fbFilterWeight2(
				rIn:=				DINT_TO_REAL(InWeight2Value), 
				tTimeConstant:= 	T#25MS, //bylo 25
				rOut=>				rFilteredWeight2Value);
				
fbFilterWeight3(
				rIn:=				DINT_TO_REAL(InWeight3Value), 
				tTimeConstant:= 	T#52MS, //bylo 25
				rOut=>				rFilteredWeight3Value);
				
fbFilterWeight4(
				rIn:=				DINT_TO_REAL(InWeight4Value), 
				tTimeConstant:= 	T#25MS, //bylo 25
				rOut=>				rFilteredWeight4Value);
///////////////////////////////////////////////////////////////////////////////				
fbFilterWeight5(
				rIn:=				DINT_TO_REAL(InWeight5Value), 
				tTimeConstant:= 	T#25MS, //bylo 25
				rOut=>				rFilteredWeight5Value);
								
fbFilterWeight6(
				rIn:=				DINT_TO_REAL(InWeight6Value), 
				tTimeConstant:= 	T#25MS, //bylo 25
				rOut=>				rFilteredWeight6Value);														
/////////////////////////////////////////////////////////////////////////////

tonIbWeight1FormSensor			(IN:=IbWeight1FormSensor ,		PT:=T#120MS); //160
tonIbWeight2FormSensor			(IN:=IbWeight2FormSensor ,		PT:=T#120MS); //160
tonIbWeight3FormSensor			(IN:=IbWeight3FormSensor ,		PT:=T#120MS); //160
tonIbWeight4FormSensor			(IN:=IbWeight4FormSensor ,		PT:=T#120MS); //160
tonIbWeight5FormSensor			(IN:=IbWeight5FormSensor ,		PT:=T#120MS); //60
tonIbWeight6FormSensor			(IN:=IbWeight6FormSensor ,		PT:=T#120MS); //60

IF VIS.nFormTransportersScrewerVelocitySVShow < 500 THEN
	fbIbWeight1FormBeforeSensor	(bIN:=IbWeight1ActuatorSensorUp,	tFilterTimeOn:=T#70MS,	tFilterTimeOff:=T#150MS);
	fbIbWeight2FormBeforeSensor	(bIN:=IbWeight2ActuatorSensorUp,	tFilterTimeOn:=T#70MS,	tFilterTimeOff:=T#150MS);
	fbIbWeight3FormBeforeSensor	(bIN:=IbWeight3ActuatorSensorUp,	tFilterTimeOn:=T#70MS,	tFilterTimeOff:=T#150MS);
	fbIbWeight4FormBeforeSensor	(bIN:=IbWeight4ActuatorSensorUp,	tFilterTimeOn:=T#70MS,	tFilterTimeOff:=T#150MS);
ELSE
	fbIbWeight1FormBeforeSensor	(bIN:=IbWeight1ActuatorSensorUp,	tFilterTimeOn:=T#10MS,	tFilterTimeOff:=T#10MS);//bylo 40 i 20
	fbIbWeight2FormBeforeSensor	(bIN:=IbWeight2ActuatorSensorUp,	tFilterTimeOn:=T#10MS,	tFilterTimeOff:=T#10MS);//bylo 40 i 20
	fbIbWeight3FormBeforeSensor	(bIN:=IbWeight3ActuatorSensorUp,	tFilterTimeOn:=T#10MS,	tFilterTimeOff:=T#10MS);//bylo 40 i 20
	fbIbWeight4FormBeforeSensor	(bIN:=IbWeight4ActuatorSensorUp,	tFilterTimeOn:=T#10MS,	tFilterTimeOff:=T#10MS);//bylo 40 i 20	
END_IF

IF VIS.nFormTransportersDispencerVelocitySVShow < 500 THEN
	fbIbWeight5FormBeforeSensor	(bIN:=IbWeight5FormSensor,			tFilterTimeOn:=T#70MS,	tFilterTimeOff:=T#150MS);
	fbIbWeight6FormBeforeSensor	(bIN:=IbWeight6FormSensor,			tFilterTimeOn:=T#70MS,	tFilterTimeOff:=T#150MS);
ELSE
	fbIbWeight5FormBeforeSensor	(bIN:=IbWeight5FormSensor,			tFilterTimeOn:=T#70MS,	tFilterTimeOff:=T#150MS);
	fbIbWeight6FormBeforeSensor	(bIN:=IbWeight6FormSensor,			tFilterTimeOn:=T#70MS,	tFilterTimeOff:=T#150MS);
END_IF
END_ACTION

ACTION aWeight1:
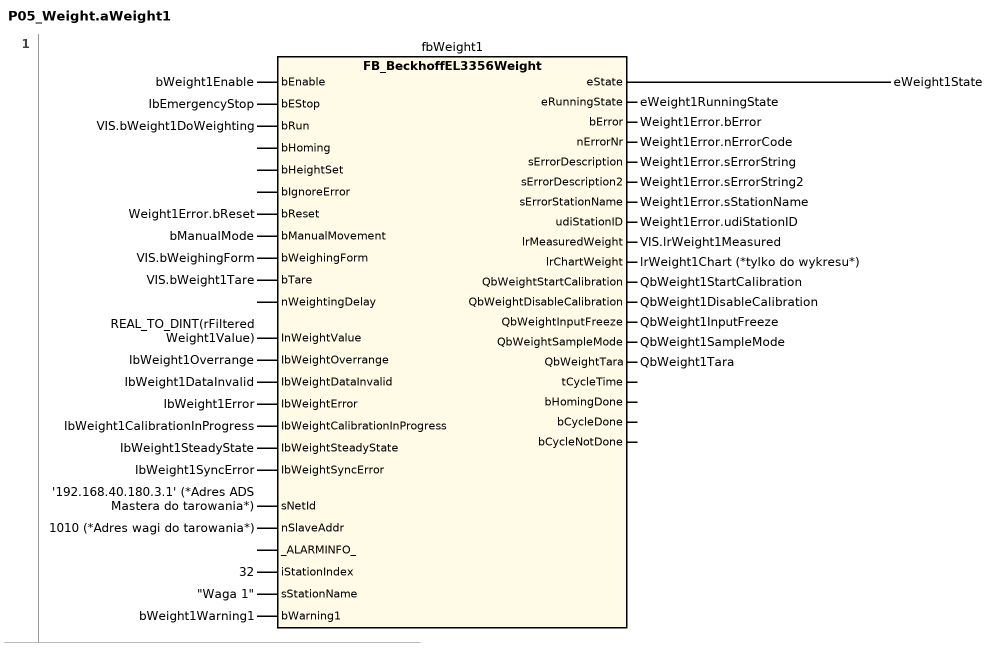
// NETWORK 1
fbWeight1(
    bEnable := bWeight1Enable,
    bEStop := IbEmergencyStop,
    bRun := VIS.bWeight1DoWeighting,
    bReset := Weight1Error.bReset,
    bManualMovement := bManualMode,
    bWeighingForm := VIS.bWeighingForm,
    bTare := VIS.bWeight1Tare,
    InWeightValue := REAL_TO_DINT(rFilteredWeight1Value),
    IbWeightOverrange := IbWeight1Overrange,
    IbWeightDataInvalid := IbWeight1DataInvalid,
    IbWeightError := IbWeight1Error,
    IbWeightCalibrationInProgress := IbWeight1CalibrationInProgress,
    IbWeightSteadyState := IbWeight1SteadyState,
    IbWeightSyncError := IbWeight1SyncError,
    sNetId := '192.168.40.180.3.1' (*Adres ADS Mastera do tarowania*),
    nSlaveAddr := 1010 (*Adres wagi do tarowania*),
    iStationIndex := 32,
    sStationName := "Waga 1",
    bWarning1 := bWeight1Warning1,
    eRunningState => eWeight1RunningState,
    bError => Weight1Error.bError,
    nErrorNr => Weight1Error.nErrorCode,
    sErrorDescription => Weight1Error.sErrorString,
    sErrorDescription2 => Weight1Error.sErrorString2,
    sErrorStationName => Weight1Error.sStationName,
    udiStationID => Weight1Error.udiStationID,
    lrMeasuredWeight => VIS.lrWeight1Measured,
    lrChartWeight => lrWeight1Chart (*tylko do wykresu*),
    QbWeightStartCalibration => QbWeight1StartCalibration,
    QbWeightDisableCalibration => QbWeight1DisableCalibration,
    QbWeightInputFreeze => QbWeight1InputFreeze,
    QbWeightSampleMode => QbWeight1SampleMode,
    QbWeightTara => QbWeight1Tara); // FB_BeckhoffEL3356Weight
eWeight1State := fbWeight1.eState;
END_ACTION

ACTION aWeight2:
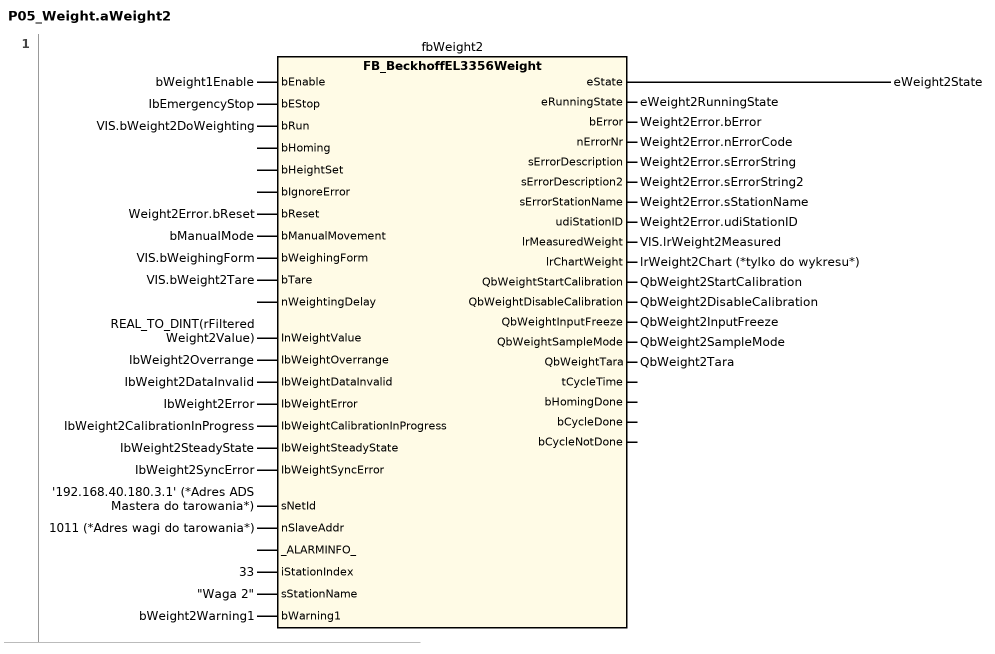
// NETWORK 1
fbWeight2(
    bEnable := bWeight1Enable,
    bEStop := IbEmergencyStop,
    bRun := VIS.bWeight2DoWeighting,
    bReset := Weight2Error.bReset,
    bManualMovement := bManualMode,
    bWeighingForm := VIS.bWeighingForm,
    bTare := VIS.bWeight2Tare,
    InWeightValue := REAL_TO_DINT(rFilteredWeight2Value),
    IbWeightOverrange := IbWeight2Overrange,
    IbWeightDataInvalid := IbWeight2DataInvalid,
    IbWeightError := IbWeight2Error,
    IbWeightCalibrationInProgress := IbWeight2CalibrationInProgress,
    IbWeightSteadyState := IbWeight2SteadyState,
    IbWeightSyncError := IbWeight2SyncError,
    sNetId := '192.168.40.180.3.1' (*Adres ADS Mastera do tarowania*),
    nSlaveAddr := 1011 (*Adres wagi do tarowania*),
    iStationIndex := 33,
    sStationName := "Waga 2",
    bWarning1 := bWeight2Warning1,
    eRunningState => eWeight2RunningState,
    bError => Weight2Error.bError,
    nErrorNr => Weight2Error.nErrorCode,
    sErrorDescription => Weight2Error.sErrorString,
    sErrorDescription2 => Weight2Error.sErrorString2,
    sErrorStationName => Weight2Error.sStationName,
    udiStationID => Weight2Error.udiStationID,
    lrMeasuredWeight => VIS.lrWeight2Measured,
    lrChartWeight => lrWeight2Chart (*tylko do wykresu*),
    QbWeightStartCalibration => QbWeight2StartCalibration,
    QbWeightDisableCalibration => QbWeight2DisableCalibration,
    QbWeightInputFreeze => QbWeight2InputFreeze,
    QbWeightSampleMode => QbWeight2SampleMode,
    QbWeightTara => QbWeight2Tara); // FB_BeckhoffEL3356Weight
eWeight2State := fbWeight2.eState;
END_ACTION

ACTION aWeight3:
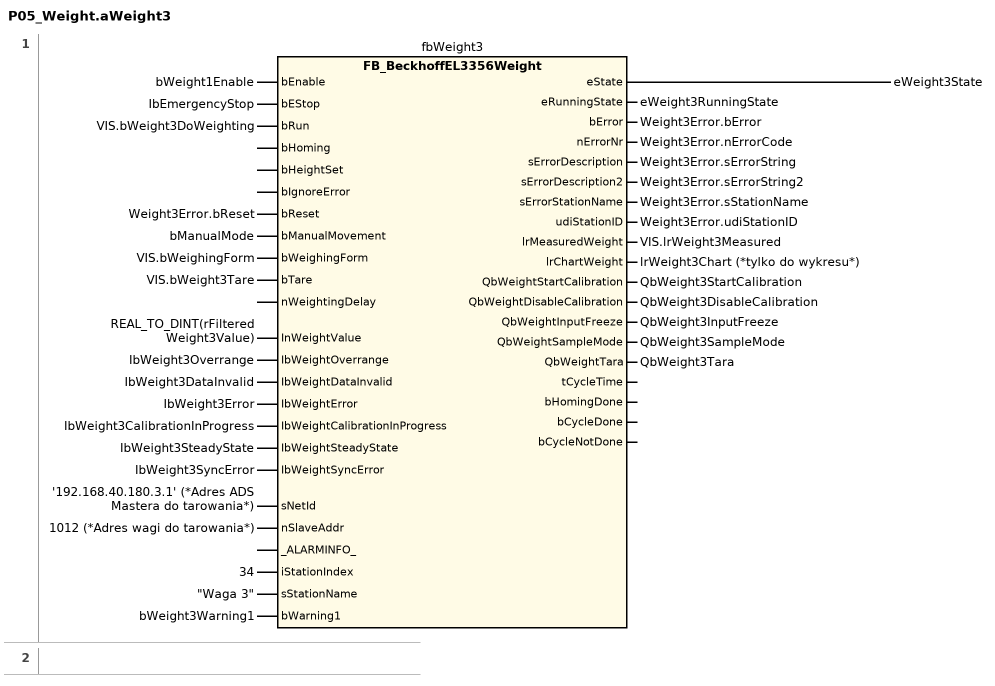
// NETWORK 1
fbWeight3(
    bEnable := bWeight1Enable,
    bEStop := IbEmergencyStop,
    bRun := VIS.bWeight3DoWeighting,
    bReset := Weight3Error.bReset,
    bManualMovement := bManualMode,
    bWeighingForm := VIS.bWeighingForm,
    bTare := VIS.bWeight3Tare,
    InWeightValue := REAL_TO_DINT(rFilteredWeight3Value),
    IbWeightOverrange := IbWeight3Overrange,
    IbWeightDataInvalid := IbWeight3DataInvalid,
    IbWeightError := IbWeight3Error,
    IbWeightCalibrationInProgress := IbWeight3CalibrationInProgress,
    IbWeightSteadyState := IbWeight3SteadyState,
    IbWeightSyncError := IbWeight3SyncError,
    sNetId := '192.168.40.180.3.1' (*Adres ADS Mastera do tarowania*),
    nSlaveAddr := 1012 (*Adres wagi do tarowania*),
    iStationIndex := 34,
    sStationName := "Waga 3",
    bWarning1 := bWeight3Warning1,
    eRunningState => eWeight3RunningState,
    bError => Weight3Error.bError,
    nErrorNr => Weight3Error.nErrorCode,
    sErrorDescription => Weight3Error.sErrorString,
    sErrorDescription2 => Weight3Error.sErrorString2,
    sErrorStationName => Weight3Error.sStationName,
    udiStationID => Weight3Error.udiStationID,
    lrMeasuredWeight => VIS.lrWeight3Measured,
    lrChartWeight => lrWeight3Chart (*tylko do wykresu*),
    QbWeightStartCalibration => QbWeight3StartCalibration,
    QbWeightDisableCalibration => QbWeight3DisableCalibration,
    QbWeightInputFreeze => QbWeight3InputFreeze,
    QbWeightSampleMode => QbWeight3SampleMode,
    QbWeightTara => QbWeight3Tara); // FB_BeckhoffEL3356Weight
eWeight3State := fbWeight3.eState;

// NETWORK 2
END_ACTION

ACTION aWeight4:
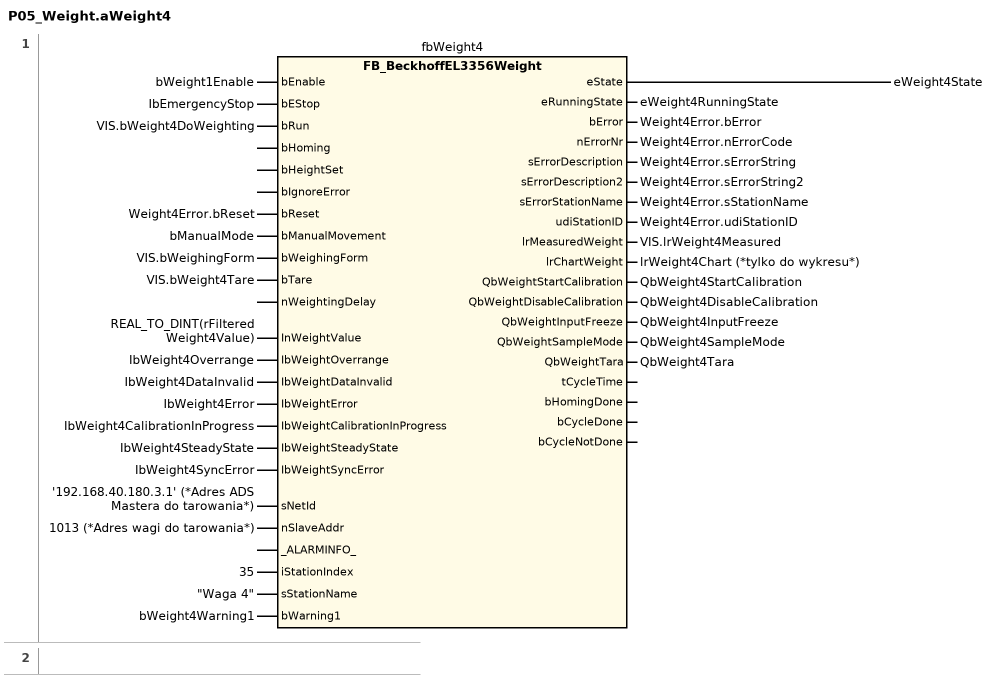
// NETWORK 1
fbWeight4(
    bEnable := bWeight1Enable,
    bEStop := IbEmergencyStop,
    bRun := VIS.bWeight4DoWeighting,
    bReset := Weight4Error.bReset,
    bManualMovement := bManualMode,
    bWeighingForm := VIS.bWeighingForm,
    bTare := VIS.bWeight4Tare,
    InWeightValue := REAL_TO_DINT(rFilteredWeight4Value),
    IbWeightOverrange := IbWeight4Overrange,
    IbWeightDataInvalid := IbWeight4DataInvalid,
    IbWeightError := IbWeight4Error,
    IbWeightCalibrationInProgress := IbWeight4CalibrationInProgress,
    IbWeightSteadyState := IbWeight4SteadyState,
    IbWeightSyncError := IbWeight4SyncError,
    sNetId := '192.168.40.180.3.1' (*Adres ADS Mastera do tarowania*),
    nSlaveAddr := 1013 (*Adres wagi do tarowania*),
    iStationIndex := 35,
    sStationName := "Waga 4",
    bWarning1 := bWeight4Warning1,
    eRunningState => eWeight4RunningState,
    bError => Weight4Error.bError,
    nErrorNr => Weight4Error.nErrorCode,
    sErrorDescription => Weight4Error.sErrorString,
    sErrorDescription2 => Weight4Error.sErrorString2,
    sErrorStationName => Weight4Error.sStationName,
    udiStationID => Weight4Error.udiStationID,
    lrMeasuredWeight => VIS.lrWeight4Measured,
    lrChartWeight => lrWeight4Chart (*tylko do wykresu*),
    QbWeightStartCalibration => QbWeight4StartCalibration,
    QbWeightDisableCalibration => QbWeight4DisableCalibration,
    QbWeightInputFreeze => QbWeight4InputFreeze,
    QbWeightSampleMode => QbWeight4SampleMode,
    QbWeightTara => QbWeight4Tara); // FB_BeckhoffEL3356Weight
eWeight4State := fbWeight4.eState;

// NETWORK 2
END_ACTION

ACTION aWeight5:
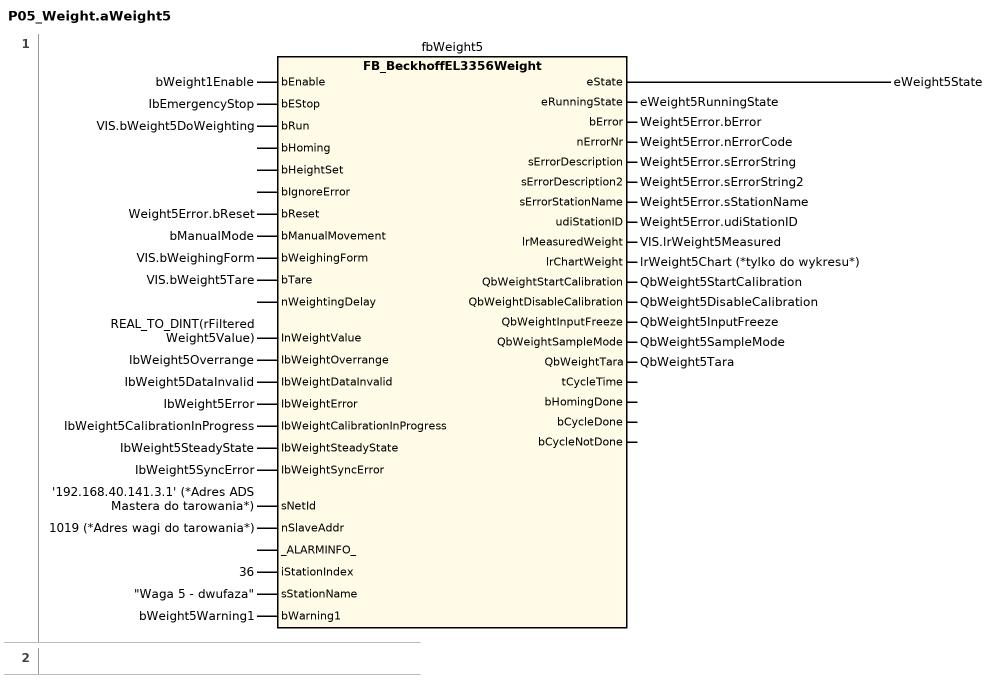
// NETWORK 1
fbWeight5(
    bEnable := bWeight1Enable,
    bEStop := IbEmergencyStop,
    bRun := VIS.bWeight5DoWeighting,
    bReset := Weight5Error.bReset,
    bManualMovement := bManualMode,
    bWeighingForm := VIS.bWeighingForm,
    bTare := VIS.bWeight5Tare,
    InWeightValue := REAL_TO_DINT(rFilteredWeight5Value),
    IbWeightOverrange := IbWeight5Overrange,
    IbWeightDataInvalid := IbWeight5DataInvalid,
    IbWeightError := IbWeight5Error,
    IbWeightCalibrationInProgress := IbWeight5CalibrationInProgress,
    IbWeightSteadyState := IbWeight5SteadyState,
    IbWeightSyncError := IbWeight5SyncError,
    sNetId := '192.168.40.141.3.1' (*Adres ADS Mastera do tarowania*),
    nSlaveAddr := 1019 (*Adres wagi do tarowania*),
    iStationIndex := 36,
    sStationName := "Waga 5 - dwufaza",
    bWarning1 := bWeight5Warning1,
    eRunningState => eWeight5RunningState,
    bError => Weight5Error.bError,
    nErrorNr => Weight5Error.nErrorCode,
    sErrorDescription => Weight5Error.sErrorString,
    sErrorDescription2 => Weight5Error.sErrorString2,
    sErrorStationName => Weight5Error.sStationName,
    udiStationID => Weight5Error.udiStationID,
    lrMeasuredWeight => VIS.lrWeight5Measured,
    lrChartWeight => lrWeight5Chart (*tylko do wykresu*),
    QbWeightStartCalibration => QbWeight5StartCalibration,
    QbWeightDisableCalibration => QbWeight5DisableCalibration,
    QbWeightInputFreeze => QbWeight5InputFreeze,
    QbWeightSampleMode => QbWeight5SampleMode,
    QbWeightTara => QbWeight5Tara); // FB_BeckhoffEL3356Weight
eWeight5State := fbWeight5.eState;

// NETWORK 2
END_ACTION

ACTION aWeight6:
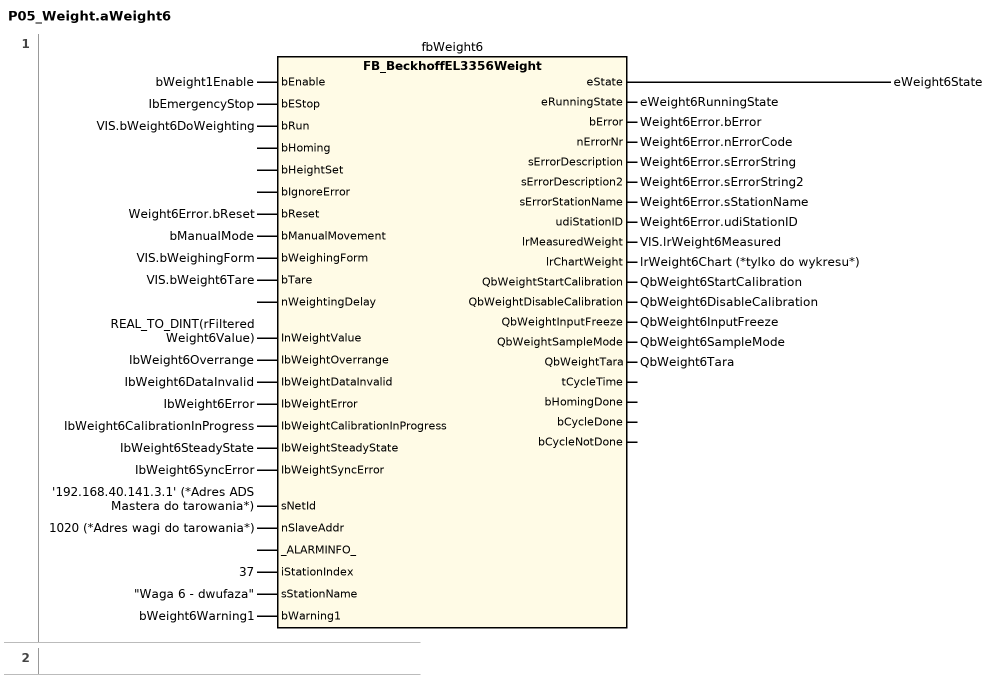
// NETWORK 1
fbWeight6(
    bEnable := bWeight1Enable,
    bEStop := IbEmergencyStop,
    bRun := VIS.bWeight6DoWeighting,
    bReset := Weight6Error.bReset,
    bManualMovement := bManualMode,
    bWeighingForm := VIS.bWeighingForm,
    bTare := VIS.bWeight6Tare,
    InWeightValue := REAL_TO_DINT(rFilteredWeight6Value),
    IbWeightOverrange := IbWeight6Overrange,
    IbWeightDataInvalid := IbWeight6DataInvalid,
    IbWeightError := IbWeight6Error,
    IbWeightCalibrationInProgress := IbWeight6CalibrationInProgress,
    IbWeightSteadyState := IbWeight6SteadyState,
    IbWeightSyncError := IbWeight6SyncError,
    sNetId := '192.168.40.141.3.1' (*Adres ADS Mastera do tarowania*),
    nSlaveAddr := 1020 (*Adres wagi do tarowania*),
    iStationIndex := 37,
    sStationName := "Waga 6 - dwufaza",
    bWarning1 := bWeight6Warning1,
    eRunningState => eWeight6RunningState,
    bError => Weight6Error.bError,
    nErrorNr => Weight6Error.nErrorCode,
    sErrorDescription => Weight6Error.sErrorString,
    sErrorDescription2 => Weight6Error.sErrorString2,
    sErrorStationName => Weight6Error.sStationName,
    udiStationID => Weight6Error.udiStationID,
    lrMeasuredWeight => VIS.lrWeight6Measured,
    lrChartWeight => lrWeight6Chart (*tylko do wykresu*),
    QbWeightStartCalibration => QbWeight6StartCalibration,
    QbWeightDisableCalibration => QbWeight6DisableCalibration,
    QbWeightInputFreeze => QbWeight6InputFreeze,
    QbWeightSampleMode => QbWeight6SampleMode,
    QbWeightTara => QbWeight6Tara); // FB_BeckhoffEL3356Weight
eWeight6State := fbWeight6.eState;

// NETWORK 2
END_ACTION

END_PROGRAM

// ---- POUs/FB/FB_BeckhoffEL3356Weight.TcPOU
(*
Nazwa:			FB_BeckhoffEL3356Weight
Opis:			Obsługa wagi
Wersja:			v0.1
Data:			2019-10-09
Autor:			DP
Urzadzenia:		waga Beckhoff
Konfiguracja:	
Info: 
- podlaczenie po module EL3356-0010
Nastawy modułu "Settings" 
Mode of operation: Standard (INT32)
RMB DATA 
Zaznaczone tylko 
	-Mode0 Filter enable: Dynamic IIR z wartością 0.2
	-Symetric reference potential active
Kalibracja zrobionia z jakaś wagą np 1kg, to wpisane 10000
Gain:1,Rated Output 0.062372, ZeroBalance 0.0209,
ScaleFactor:1, SteadyStateWindow:100ms, CalibrationInterwal:180s
SteadyStateTolerance:10,TestInteval:10,

*)


FUNCTION_BLOCK FB_BeckhoffEL3356Weight
VAR_INPUT
	bEnable: BOOL;						//Zezwolenie na pracę
	bEStop:BOOL;						//Stop Awaryjny włączony
	bRun:BOOL;							//Rozkaz łapania 
	bHoming:BOOL;						//Zezwolenie na wykonanie bazowania i pozycjonowania podajnika
	bHeightSet:BOOL;					//Ustaw wysokość
	bIgnoreError:BOOL;					//Ignorowania błędów cyklu pracy
	bReset:BOOL;						//Reset błędu, jeśli w stanie "eError"
	bManualMovement:BOOL;				//Zezwolenie na ruchy ręcznę
	bWeighingForm: BOOL;				//Wlaczone przewazanie, dluzsze czasy		
	bTare:BOOL;							//Tarowanie Wagi
	nWeightingDelay:UINT;				//Opoźnienie ważenia
	InWeightValue: DINT;				// Wartość wagi
	IbWeightOverrange: BOOL;						
	IbWeightDataInvalid: BOOL;		
	IbWeightError: BOOL;	
	IbWeightCalibrationInProgress: BOOL;
	IbWeightSteadyState: BOOL;
	IbWeightSyncError: BOOL;	
	sNetId:STRING;
	nSlaveAddr:UINT;
	
	_ALARMINFO_ :BOOL;
	iStationIndex:UDINT;					//Numer stacji 
	sStationName:WSTRING;					//Nazwa stacji	

END_VAR
VAR_OUTPUT
	eState: E_Station;						//Stan ogólny bloku
	eRunningState: E_WeightState;			//Stan wewnętrzny
	bError: BOOL;							//Błąd stacji
	nErrorNr: UDINT;						//Nr błędu podajnika platynek
	sErrorDescription:STRING;				//Opis błędu
	sErrorDescription2: STRING;				//Opis błędu 2
	sErrorStationName:STRING;				//Nazwa stacji
	udiStationID:UDINT;						// Nr stacji

	lrMeasuredWeight: LREAL; 				//Zmierzona waga 
	lrChartWeight: LREAL; 					//Zmierzona waga do wykresu
	QbWeightStartCalibration: BOOL;
	QbWeightDisableCalibration: BOOL;
	QbWeightInputFreeze: BOOL;
	QbWeightSampleMode: BOOL;
	QbWeightTara: BOOL;
	tCycleTime:TIME;
	bHomingDone:BOOL;						//Wymagane ponowne bazowanie (blad podczas bazowania lub stop awaryjny)
	bCycleDone:BOOL;
	bCycleNotDone:BOOL;
END_VAR
VAR
	(*Opóźnianie ważenia*)
	tonWeightingDelay: TON;
	
	(*Tarowanie*)
	rtrigTare: R_TRIG;
	
	(*Statystyki*)
	rtrigCycleTimerRead: R_TRIG;
	tonCycleTimer: TON;
	
	(*Próbkowanie wagi*)
	lrMeasuredWeightSampling: LREAL;
	lrWeightSampling: LREAL;
	tonWeightingDoneIfNotSteadyState: TON;
	nWeightingDoneIfNotSteadyState: INT; //Licznik ilości prawdopodobnie błędnych pomiarów
	tonWeightingDoneIfNotSteadyStateReset: TON; // Do resetowania błędu ilości błędnych pomiarów
	//
	tonOverrange	:TON;
	tonError		:TON;	
	
	(*TAROWANIE EEPROM*)
	fbCoE:FB_EcCoESdoWrite;
	wCoeData:WORD;

	nWarCheck1: INT;
	nWarCheck2: INT;
	bMinMaxAvg: BOOL;
	lrMeasuredWeightMax: LREAL;
	lrMeasuredWeightMin: LREAL;

	eLastState: E_Station;							//Stan ogólny bloku
	eLastRunningState: E_WeightState;			//Stan podbloku
	eLastStateTemp: E_Station;						//Stan ogólny bloku
	eLastRunningStateTemp: E_WeightState;		//Stan podbloku
	bStateError: BOOL;
	
	fbCalibrationDisableOff	: FB_InputFilter;

	tWeightingTime: TIME;
	
	//Zmienne od EVENTLOGGER
	bAlarmInit 						: BOOL := TRUE; 
	nAlarmNumerator					: INT;
	arfbAlarm						: ARRAY[0..19] OF  FB_TcAlarm;		//Tablica bloczków błędów
	fbSourceInfo 					: FB_TcSourceInfo;
	iSourceInfo						: I_TcSourceInfo;
	sAlarmTest						: STRING;
	tonEventLogger					: TON;
	//Koniec zmiennych od EVENTLOGGER
END_VAR

VAR_IN_OUT
	bWarning1: BOOL;		//Ostrzezenie przed brakiem stabilizacji wagi
END_VAR

aWeighingForm();
ErrorHandling();
Control();
Statistics();
aStationID();

(*Zapisywanie ostatniego stanu*)
IF eLastStateTemp<>eState THEN
	eLastState := eLastStateTemp;
END_IF
eLastStateTemp := eState;
IF eLastRunningStateTemp<>eRunningState THEN
	eLastRunningState := eLastRunningStateTemp;
END_IF
eLastRunningStateTemp := eRunningState;
(*Koniec Zapisywanie ostatniego stanu*)

//do testów, bo co 180s robi samokalibracje!
fbCalibrationDisableOff(bIN:=bRun, tFilterTimeOn:=T#10MS, tFilterTimeOff:=T#2S);
IF fbCalibrationDisableOff.bOUT THEN
	QbWeightDisableCalibration:=TRUE;
ELSE 
	QbWeightDisableCalibration:=FALSE;
	
END_IF
//QbWeightTara:=bTare;

ACTION aStationID:
udiStationID	:=	iStationIndex;
END_ACTION

ACTION aWeighingForm:
(*
IF bWeighingForm THEN //Wlaczone przewazanie formatek
	nWeightingDelay := 2000; //Opoznienie przed wazeniem
	tWeightingTime	:= T#800MS; //Czas ważenia
ELSE				// Wylaczone przewazanie
	tWeightingTime := T#500MS; //Czas ważenia
END_IF
*)





IF bWeighingForm THEN //Wlaczone przewazanie formatek
	nWeightingDelay := 685;//685 //Opoznienie przed wazeniem
	tWeightingTime	:= T#300MS;//T#150MS; //Czas ważenia
ELSE				// Wylaczone przewazanie
	tWeightingTime := T#150MS;//T#150MS; //Czas ważenia
	//tWeightingTime := T#100MS;//T#490MS;//T#500MS; //Czas ważenia	
END_IF
END_ACTION

ACTION Control:

	(** TIMERY**)
	//Opóźnienie ważenia, trzeba tutaj uwzględnić jeszcze czas ustawiania bitu SteadyState
	tonWeightingDelay(IN:=(eRunningState=E_WeightState.eWeighting), PT:=UINT_TO_TIME(nWeightingDelay));
	//Jeżeli nie ma stabilizacji wagi to po tym czasie podaj pomiar z próbkowania
	tonWeightingDoneIfNotSteadyState(IN:=eRunningState=E_WeightState.eWeighting AND tonWeightingDelay.Q, PT:=tWeightingTime); //bylo 550

	(*****Wyłączenie enable*****)
	IF NOT bEnable THEN
		IF eState <> E_Station.eDisabled AND eState <> E_Station.ePreparingToDisable THEN
				eState 				:= E_Station.ePreparingToDisable; 
		END_IF	
	END_IF

	(*****Estop*****)
	IF NOT bEstop  THEN	
		IF eState <> E_Station.eAborted AND eState <> E_Station.eAborting AND eState <> E_Station.eDisabled THEN
				eState 				:= E_Station.eAborting; 
		END_IF
	END_IF

	CASE eState OF
	/////////////////////////////	
		E_Station.eDisabled: 					// Stan nieaktywnosci (Stacja wyłączona) 

			IF bEnable THEN
				eState 				:= E_Station.ePreparingToReady; 
			END_IF 
			
    /////////////////////////////	    
		E_Station.eAborted: 					// Stan bezpiecznego zatrzymania (po Abortingu) 

			IF bEStop THEN
				eState 				:= E_Station.ePreparingToReady;
			END_IF
			
	/////////////////////////////	
		E_Station.eAborting:                 	// Stan bezpiecznego zatrzymywania (po EStopie)

		
			eState := E_Station.eAborted;  
			eRunningState:=E_WeightState.eDisabled;
			
	/////////////////////////////			
		E_Station.eError:                 	 	// Stan błędu 	

			IF bReset THEN
				eState 				:= E_Station.eResetting;
				
			END_IF
						
	/////////////////////////////
		E_Station.eResetting:					// Stan resetowania bledu (po Errorze)
	
			bError := FALSE;

			IF NOT bError THEN
				nErrorNr 			:=	0;
   				sErrorDescription 	:=	'';
				eState 				:=	E_Station.ePreparingToReady;
			ELSE
				eState 				:=	E_Station.eError;
			END_IF
        
	/////////////////////////////
		E_Station.eManualMovement:     			// Stan ruchów manualnych  

			ManualMovements();
			//Wyjście z trybu serwisowego
			IF NOT bManualMovement THEN
				eState:=E_Station.eReady;
			END_IF

	/////////////////////////////
		E_Station.eHoming:						// Stan bazowania 

			Homing();
			IF NOT bHoming AND NOT bHeightSet THEN
			   eState:=E_Station.ePreparingToReady;
			END_IF		
			
	/////////////////////////////
		E_Station.eHomingDone:                  // Stan wykonania bazowania 
	
			bHomingDone							:=	TRUE;
			IF NOT bHoming AND NOT bHeightSet THEN
			   eState:=E_Station.eReady;
			END_IF
			
	/////////////////////////////
		E_Station.ePreparingToReady:            // Stan przygotowywania do gotowosci (zawsze przed Ready)  
	
			eRunningState:=E_WeightState.eReady;
			eState:=E_Station.eReady;	
			
	/////////////////////////////
		E_Station.ePreparingToDisable:          // Stan przygotowywania do nieaktywnosci (po wyłączeniu Enable) 
  
			eState:=E_Station.eDisabled;
			eRunningState:=E_WeightState.eDisabled;

				
	/////////////////////////////
		E_Station.eReady:						// Stan gotowosci 

			IF bRun AND NOT bCycleDone AND NOT bCycleNotDone THEN
				eState 				:= E_Station.eStarting; 
			END_IF
			IF bHoming OR bHeightSet THEN
				eState 				:= E_Station.eHoming; 
			END_IF
			IF bManualMovement THEN
				//Jeśli przejście w tryb ruchów manualnych przepisz wszystkie stany siłowników sterowanych przez moduł
				//aby zapobiec ewentualnym kolizjom po wejściu w tryb serwisowy
				
				eState 						:= E_Station.eManualMovement; 
				eRunningState 				:= E_WeightState.eReady;
 
			END_IF
			IF NOT bRun THEN
				bCycleDone 			:= FALSE;
				bCycleNotDone 		:= FALSE;			
			END_IF
			
	/////////////////////////////
		E_Station.eStopping:					// Stan zatrzymywania 
					
			Running();
			(*IF bOpenedActuatorSensor THEN*)
				eState	:=	E_Station.eReady;
			(*END_IF*)
			
	/////////////////////////////
		E_Station.eStarting:                  	// Stan uruchamiania (po Ready)
				
			eState					 := E_Station.eRunning; 

	/////////////////////////////
		E_Station.eRunning:               		// Stan wykonywania cyklu (po Startingu), w tym stanie osobny

			Running();
			IF NOT bRun THEN 					(*Przerywanie cyklu*)
				eState				:= E_Station.eStopping;
				bCycleNotDone		:= TRUE;
			END_IF
			IF bCycleDone OR bCycleNotDone THEN (*Cykl zakończony*)
				eState 				 := E_Station.eReady;
			END_IF						
		ELSE
		
		
	/////////////////////////////		
	END_CASE
END_ACTION

ACTION ErrorHandling:
// Alarm_0320	320	Error	Błąd modułu - sprawdź połączenie
// Alarm_0321	321	Error	Przekroczenie zakresu - sprawdź czy nie jest zablokowana
IF bAlarmInit THEN
    bAlarmInit := FALSE; 
	fbSourceInfo.Clear();
	fbSourceInfo.sName:=wsLiteral_TO_UTF8(sStationName);//'Machine';
	fbSourceInfo.nId:=udiStationID;//2700;
	// Alarm_0320	320	Error	Błąd modułu - sprawdź połączenie
    arfbAlarm[0].CreateEx(stEventEntry := TC_EVENTS.AlarmClass.Alarm_0320, bWithConfirmation:= FALSE,  ipSourceInfo:= fbSourceInfo); 
	// Alarm_0321	321	Error	Przekroczenie zakresu - sprawdź czy nie jest zablokowana
	arfbAlarm[1].CreateEx(stEventEntry := TC_EVENTS.AlarmClass.Alarm_0321, bWithConfirmation:= FALSE,  ipSourceInfo:= fbSourceInfo);
END_IF

//OBSŁUGA BŁĘDÓW PODAJNIKA PLATYNEK

//************LISTA BŁĘDÓW***************
bStateError:= (eState=E_Station.eError) OR (eState=E_Station.eResetting) OR bIgnoreError;
tonEventLogger (IN:= NOT tonEventLogger.Q, PT:=T#1S);

IF tonEventLogger.Q THEN
	IF bEnable THEN
		// Alarm_0320	320	Error	Błąd modułu - sprawdź połączenie
		//Error 1 - Bład modułu wagi
		tonError(IN:=IbWeightError,	PT:=T#1S);	
		IF tonError.Q AND NOT bStateError THEN
			IF NOT arfbAlarm[0].bActive THEN
				//bRun:=FALSE;
				arfbAlarm[0].Raise(nTimeStamp:=0);
			END_IF
		ELSE	
			IF  arfbAlarm[0].bActive AND bReset THEN
				arfbAlarm[0].Clear(nTimeStamp:=0, bResetConfirmation:= FALSE);
			END_IF	
	//		bRun:=FALSE;
	// 		sErrorDescription:='Błąd modułu - sprawdź połączenie';
	// 		sErrorDescription2:='';
	// 		bError := TRUE;
	// 		nErrorNr:=201;	
			//nErrorNr := nErrorNr+iStationIndex;
		END_IF
	
		//Error 2 - Brak stabilizacji wagi
		tonWeightingDoneIfNotSteadyStateReset(IN:=nWeightingDoneIfNotSteadyState>0, PT:=T#10S);  (*Jeżeli przez więcej niż 1 min nie osiągnelo 10 pomiarów to resetuj*)
		IF tonWeightingDoneIfNotSteadyStateReset.Q THEN 
				nWeightingDoneIfNotSteadyState:=0; 
				bWarning1 := FALSE;
				nWarCheck1:=nWarCheck1+1;
		END_IF	
		IF nWeightingDoneIfNotSteadyState>10 AND NOT bWarning1 THEN
			bWarning1 := TRUE;
			nWarCheck2:=nWarCheck2+1;
		END_IF;
		// Alarm_0321	321	Error	Przekroczenie zakresu - sprawdź czy nie jest zablokowana
		//Error 3 - BłPrzekroczono poziom pomiarowy
		tonOverrange(IN:=IbWeightOverrange,	PT:=T#1S);
		IF tonOverrange.Q AND NOT bStateError THEN
			IF NOT arfbAlarm[1].bActive THEN
				arfbAlarm[1].Raise(nTimeStamp:=0);
			END_IF
		ELSE	
			IF  arfbAlarm[1].bActive AND bReset THEN
				arfbAlarm[1].Clear(nTimeStamp:=0, bResetConfirmation:= FALSE);
			END_IF	
			//bRun:=FALSE;
	// 		bError := TRUE;
	// 		nErrorNr:=202;
	// 		//nErrorNr := nErrorNr+iStationIndex;
	// 		sErrorDescription:='Przekroczenie zakresu - sprawdź czy nie jest zablokowana';	
	// 		sErrorDescription2:='';			
		END_IF
	
	ELSE
		bError := FALSE;
	END_IF
		
		
	//******************PRZEJŚCIE DO eERROR*****************************

	IF bError AND NOT bStateError THEN
		IF eLastState = eRunning THEN
			bCycleNotDone := TRUE;
		END_IF
		eState := E_Station.eError;
	END_IF
	
	//****************WYŚWIETLANIE STATUSU BLEDU***********************
	
	(*Wyświetlanie błedu na wyjściu*)
	bError							:= FALSE;
	FOR nAlarmNumerator := 0 TO 19 DO
		bError						:= bError OR arfbAlarm[nAlarmNumerator].bActive;
	END_FOR
	
END_IF

(*Przepisywanie nazwy stacji*)
sErrorStationName := WSTRING_TO_STRING(sStationName);
END_ACTION

ACTION Homing:
//BAZOWANIE

eState:=E_Station.eHomingDone;
END_ACTION

ACTION ManualMovements:

//W trybie ruchów manualnych wykonuj ruchy za pomocą rozkazów manualnych
Running();


IF NOT bRun THEN
	bCycleDone 					:= FALSE;
	bCycleNotDone 				:= FALSE;	
END_IF
END_ACTION

ACTION Running:

CASE eRunningState OF
	
	//NIEGOTOWY
	E_WeightState.eDisabled:
		IF bEnable THEN
			eRunningState:=E_WeightState.eReady;
		END_IF
		
	//WAGA GOTOWA DO PRACY
	E_WeightState.eReady: 
		//Jeśli komenda chwytania przejdz do stanu chwytanie
		IF NOT bCycleDone AND NOT bCycleNotDone THEN
			IF bRun THEN
				eRunningState:=E_WeightState.eWeighting;
			END_IF
		END_IF
		rtrigTare(CLK:=bTare,Q=>);
			
			(*IF rtrigTare.Q THEN
				QbWeightTara:=TRUE;
			ELSE
				QbWeightTara:=FALSE;
			END_IF*)
			
			(*Tarowanie EEPROM*)
			wCoeData := 16#0002; (* tara EEProm*)
			fbCoE(
				sNetId		:= sNetId,
				nSlaveAddr 	:= nSlaveAddr,
				nSubIndex 	:= 16#01,
				nIndex 		:= 16#FB00,
				pSrcBuf 	:= ADR(wCoeData),
				cbBufLen 	:= SIZEOF(wCoeData),
				bExecute 	:= rtrigTare.Q,
				tTimeout 	:= t#5s
			);
		lrMeasuredWeightSampling := lrWeightSampling := 0; 		(*Kasowanie zmiennych od próbkowania*)
		lrMeasuredWeightMin := lrMeasuredWeightMax := 0;

			QbWeightTara:=bTare;

	///WAGA W STANIE WAŻENIA
	E_WeightState.eWeighting:
		IF tonWeightingDelay.Q AND IbWeightSteadyState (*AND TEST*) THEN		(*Czekanie na sygnał stabilizacji z modułu wagi*)
			lrMeasuredWeight := DINT_TO_REAL(InWeightValue)/10.0;
			eRunningState:=E_WeightState.eWeightingDone;
		ELSIF tonWeightingDelay.Q THEN							(*Jeżeli nie ma sygnału to zaczynaj próbokować wagę co cykl*)
			IF bMinMaxAvg THEN
				lrMeasuredWeightSampling := DINT_TO_REAL(InWeightValue)/10.0;
				
				IF	lrMeasuredWeightMin = 0 THEN
					lrMeasuredWeightMin := lrMeasuredWeightSampling;
				END_IF

				IF lrMeasuredWeightSampling > lrMeasuredWeightMax THEN
					lrMeasuredWeightMax := lrMeasuredWeightSampling;
				END_IF
				IF lrMeasuredWeightSampling < lrMeasuredWeightMin THEN
					lrMeasuredWeightMin := lrMeasuredWeightSampling;
				END_IF
				IF tonWeightingDoneIfNotSteadyState.Q THEN
					lrMeasuredWeight := (lrMeasuredWeightMax + lrMeasuredWeightMin)/2; (*Podaj pmiar z próbokowania jeżeli nie było stabilizacji*)
					eRunningState:=E_WeightState.eWeightingDone;
				END_IF
				
				
			ELSE	
				lrMeasuredWeightSampling :=lrMeasuredWeightSampling + DINT_TO_REAL(InWeightValue)/10.0;
				lrWeightSampling := lrWeightSampling + 1 ;
				IF tonWeightingDoneIfNotSteadyState.Q THEN
					lrMeasuredWeight := lrMeasuredWeightSampling / lrWeightSampling; (*Podaj pmiar z próbokowania jeżeli nie było stabilizacji*)
					eRunningState:=E_WeightState.eWeightingDone;
					nWeightingDoneIfNotSteadyState := nWeightingDoneIfNotSteadyState +1 ;
				END_IF	
			END_IF
				
		END_IF		
		
		//ZWAŻONO
	E_WeightState.eWeightingDone:

		bCycleDone := TRUE;
		eRunningState:=E_WeightState.eReady;
		//Kiedy zniknie rozkaz chwytania i 

END_CASE
END_ACTION

ACTION Statistics:
rtrigCycleTimerRead(CLK:=eRunningState=E_WeightState.eWeightingDone);
IF rtrigCycleTimerRead.Q THEN
	tCycleTime:=tonCycleTimer.ET;
END_IF
tonCycleTimer(IN:=eRunningState>E_WeightState.eReady,PT:=T#1D);
END_ACTION

END_FUNCTION_BLOCK

// ---- POUs/FB/NewFBs/FB_WeightStation.TcPOU
(*
Nazwa:		FB_WeightStation
Opis:		Podnoszenie wag
Wersja:		V0.26
Data:		04.09.2024
Autor:		DP, 
Urządzenia:	Siłowniki
Ostatnie zmiany:
	- 20250904 [DP] EventLog-do sprawdzenia, 1 spr->wywołać błędy 
	- 2024-10-01 [DP] Liczniki po Aborting
	- 2024-04-17 [DP] Przerobienie liczenia i uprowszenie, dwufaz

Konfiguracja:
	- Krokówka
	Instukcja:
		-
		-
	
Info:
	- 
*)

FUNCTION_BLOCK FB_WeightStation
VAR_INPUT
	bEnable											: BOOL;
	bEStop											: BOOL;
	bRun											: BOOL;

	bTwoPhaseMode									: BOOL;
	bCountingBeforeSensorsMode						: BOOL;
    eGlobalState        							: E_PMLState; 							//Stan ogólny maszyny, tylko do błędu
	bConveyorRunning								: BOOL;									//Transporter pracuje, tylko do błędu
	bWeight1ActuatorSensorUp						: BOOL;									//Pierwsza waga podniesiona
	bWeight1FormSensor								: BOOL;									//Obecność formatki na pierwszej wadze     
	bWeight1FormBeforeSensor						: BOOL;									//Obecność formatki przed pierwszą wagą 

	bWeight2ActuatorSensorUp						: BOOL;									//Druga waga podniesiona
	bWeight2FormSensor								: BOOL;									//Obecność formatki na drugiek wadze
	bWeight2FormBeforeSensor						: BOOL;									//Obecność formatki przed pierwszą wagą 
	
	bWeight3ActuatorSensorUp						: BOOL;									//Trzecia waga podniesiona
	bWeight3FormSensor								: BOOL;									//Obecność formatki na trzeciej wadze
	bWeight3FormBeforeSensor						: BOOL;									//Obecność formatki przed pierwszą wagą 
	
	bWeight4ActuatorSensorUp						: BOOL;									//Czwarta waga podniesiona
	bWeight4FormSensor								: BOOL;									//Obecność formatki na czwartej wadze
	bWeight4FormBeforeSensor						: BOOL;									//Obecność formatki przed pierwszą wagą 
	
	bCanReleaseForms								: BOOL;									//Można wypuścić formatki
	bWeighingCycle									: BOOL;									//Trwa ważenie
                                    	
	arrWeightPackageState							: ARRAY [1..17] OF S_PackageState;		//Rejestr nad wagami
	
	bResetCycle										: BOOL;									//Reset cyklu
	
	bHoming											: BOOL;
	bIgnoreError									: BOOL;
	bReset											: BOOL;
	bManualMovement									: BOOL;
	                                    			
	_TIMERS_										: BOOL;
	tWeight1ActuatorUpDelay							: TIME;									//Opóźnienie podnoszenia wagi 1
	tWeight2ActuatorUpDelay							: TIME;									//Opóźnienie podnoszenia wagi 2
	tWeight3ActuatorUpDelay							: TIME;									//Opóźnienie podnoszenia wagi 3
	tWeight4ActuatorUpDelay							: TIME;									//Opóźnienie podnoszenia wagi 4
	
	_ALARMINFO_										: BOOL;
	udiStationIndex									: UDINT;								//Numer stacji
	sStationName									: WSTRING;
	
END_VAR   
                              			
VAR_OUTPUT                              			
	eState											: E_Station;							//Stan ogólny bloku
	eRunningState									: E_WeightLiftStationState;				//Stan stacji
	
	bWeight1Actuator								: BOOL;									//Podnoszenie 1 wagi
	bWeight2Actuator								: BOOL;									//Podnoszenie 2 wagi
	bWeight3Actuator								: BOOL;									//Podnoszenie 3 wagi
	bWeight4Actuator								: BOOL;									//Podnoszenie 4 wagi

	iFormsCounterWeight1							: INT;									//Licznik formatek
	iFormsCounterWeight2							: INT;									//Licznik formatek na wadze 2
	iFormsCounterWeight3							: INT;									//Licznik formatek na wadze 3
	iFormsCounterWeight4							: INT;									//Licznik formatek na wadze 4
	
	bError											: BOOL;									//Błąd stacji
	udiErrorID										: UDINT;								//Numer błędu
	sErrorDescription								: STRING(255);							//Opis błędu
	sErrorDescription2								: STRING(200);							//Opis błędu
	sErrorStationName								: STRING(200);							//Nazwa stacji
	udiStationID									: UDINT;								// Nr stacji
                                    			
	tCycleTime										: TIME;									//Czas cyklu
	bHomingDone										: BOOL;									//Stacja zbazowana 
	bWeighingCycleDone								: BOOL;									//Koniec ważenia 
	bCycleDone										: BOOL;									//Cykl skończony 			
	bTareWeights									: BOOL;		
END_VAR

VAR_IN_OUT
	bManualWeight1Actuator							: BOOL;									//Tryb manualny, Waga 1 UP	
	bManualWeight2Actuator							: BOOL;									//Tryb manualny, Waga 2 UP
	bManualWeight3Actuator							: BOOL;									//Tryb manualny, Waga 3 UP
	bManualWeight4Actuator							: BOOL;									//Tryb manualny, Waga 4 UP	
	bDeparture										: BOOL;					
	bAutoTare										: BOOL;	
END_VAR

VAR
	eLastStateTemp									: E_Station;							//Ostatni stan CONTROL
	eLastState										: E_Station;							//Ostatni stan CONTROL
	eLastRunningStateTemp							: E_WeightLiftStationState;				//Ostatni stan Running
	eLastRunningState								: E_WeightLiftStationState;				//Ostatni stan Running
	eRunningStateBeforeEStop	             		: E_WeightLiftStationState;	                      			                                    		
	tonWeight1ActuatorDelay							: TON;									//TON, opóźnienie podnoszenia wagi 1
	tonWeight2ActuatorDelay							: TON;									//TON, opóźnienie podnoszenia wagi 2
	tonWeight3ActuatorDelay							: TON;									//TON, opóźnienie podnoszenia wagi 3
	tonWeight4ActuatorDelay							: TON;									//TON, opóźnienie podnoszenia wagi 4
	tonWeightAntuatorOffDelay						: TON;
	tonPreparingToReadyDelay						: TON;
	tonResetting									: TON;
	tofRunning										: TOF;
	rtResetCommands									: R_TRIG;
	tonHoming 										: TON;
	tonReadyAndRepair								: TON;					
	tonAbortedDelay									: TON;
	tonRepairDelay									: TON;									//TON, czas po którym przechodzimy do naprawy
	tonRepairOnDelay								: TON;									//TON, czas na wyjazd wszystkich formatek
	rtWeight1FormSensor								: R_TRIG;								//R_Trig, zbocze nar (przy wadze 1)
	rtWeight2FormSensor								: R_TRIG;								//R_Trig, zbocze nar (przy wadze 2)
	rtWeight3FormSensor								: R_TRIG;								//R_Trig, zbocze nar (przy wadze 3)
	rtWeight4FormSensor								: R_TRIG;								//R_Trig, zbocze nar (przy wadze 4)

	ftWeight1FormBeforeSensor						: F_TRIG;								
	ftWeight2FormBeforeSensor						: F_TRIG;								
	ftWeight3FormBeforeSensor						: F_TRIG;								
	ftWeight4FormBeforeSensor						: F_TRIG;								
	
	tonWeightsEmpty									: TON;
	toniCaseTareWeights1							: TON;
	toniCaseTareWeights2							: TON;
	
	bLastStateWeight1Actuator						: BOOL;							
	bLastStateWeight2Actuator						: BOOL;	
	bLastStateWeight3Actuator						: BOOL;	
	bLastStateWeight4Actuator						: BOOL;	
	
	bStateError										: BOOL;
	bWasAborting									: BOOL;
	
	bRepairAllRegistersAreEmpty						: BOOL;								
	
	//Błedy
	bResetCycleOn									: BOOL;
	tonWeight1ActuatorUpError 						: TON;
	tonWeight2ActuatorUpError 						: TON;
	tonWeight3ActuatorUpError 						: TON;
	tonWeight4ActuatorUpError 						: TON;
	
	//Śmiecie
	tonRepair1: TON;
	tonRepair2: TON;
	tonRepair3: TON;
	tonRepair4: TON;
	tonRepair5: TON;
	tonRepair6: TON;
	
	rtrigCycleTimerRead: R_TRIG;
	tonCycleTimer: TON;
	tt: INT;
	rtWeight3FormSensorWithDelay2: R_TRIG;

	iRepair1: INT;
	iRepair2: INT;
	iRepair3: INT;
	iRepair4: INT;
	iRepair5: INT;
	iRepair6: INT;
	
	tofRunningStopping: TOF;
	iCaseTareWeights:INT;
	
	//Zmienne od EVENTLOGGER
	bAlarmInit 						: BOOL := TRUE; 
	nAlarmNumerator					: INT;
	arfbAlarm						: ARRAY[0..19] OF  FB_TcAlarm;		//Tablica bloczków błędów
	fbSourceInfo 					: FB_TcSourceInfo;
	iSourceInfo						: I_TcSourceInfo;
	sAlarmTest						: STRING;
	tonEventLogger					: TON;
	//Koniec zmiennych od EVENTLOGGER
	bTest							: BOOL;
END_VAR

ResetAll();
ACT_ErrorHandling();
ACT_Signals();
aRepair();
ACT_Control();
ACT_Statistics();
aStationID();

IF eLastStateTemp <> eState THEN
	eLastState							:= eLastStateTemp;
END_IF
eLastStateTemp							:= eState;

IF eLastRunningStateTemp <> eRunningState THEN
	eLastRunningState					:= eLastRunningStateTemp;
END_IF
eLastRunningStateTemp					:= eRunningState;

ACTION ACT_Control:


	(*****Wyłączenie enable*****)
	IF NOT bEnable AND NOT bError THEN
		IF eState <> E_Station.eDisabled AND eState <> E_Station.ePreparingToDisable THEN
				eState 								:= E_Station.ePreparingToDisable; 
		END_IF	
	END_IF

	(*****Estop*****)
	IF NOT bEstop  THEN	
		IF eState <> E_Station.eAborted AND eState <> E_Station.eAborting AND eState <> E_Station.eDisabled THEN
				eRunningStateBeforeEStop			:= eRunningState;
				eState 								:= E_Station.eAborting; 
		END_IF
	END_IF


CASE eState OF
	
	
	E_Station.eDisabled: 					// Stan nieaktywnosci (Stacja wyłączona)
		IF bEnable THEN
			eState											:= E_Station.ePreparingToReady;
		END_IF	
	//------------------------------------------------------------------------------
	
	E_Station.eAborted: 					// Stan bezpiecznego zatrzymania (po Abortingu)			
		IF bEStop THEN
			eState											:= E_Station.ePreparingToReady;
		END_IF	
	//------------------------------------------------------------------------------
	
	E_Station.eAborting:                 	// Stan bezpiecznego zatrzymywania (po EStopie)
	
		aResetCommandsAborting();
		bWasAborting										:= TRUE;
		eState												:= E_Station.eAborted;	
		eRunningState										:= E_WeightLiftStationState.eReady;
	//------------------------------------------------------------------------------
	
	E_Station.eError:                 	 	// Stan błędu 	
	
		IF bReset THEN
			eState									:= E_Station.eResetting;	
		ELSE
			aResetCommands();
		END_IF
		
	//------------------------------------------------------------------------------

	
	E_Station.eResetting:					// Stan resetowania bledu (po Errorze)

// 		CASE udiErrorID OF 
// //		CASE udiErrorID - udiStationIndex OF 
// 			
// 			191,195: //Error 1
// 				bWeight1Actuator						:=	FALSE;
// 				bError									:=	FALSE;
// 			192,196://Error 2
// 				bWeight2Actuator						:=	FALSE;
// 				bError									:=	FALSE;	
// 			193: //Error 3
// 				bWeight3Actuator						:=	FALSE;
// 				bError									:=	FALSE;
// 			194: //Error 4
// 				bWeight4Actuator						:=	FALSE;
// 				bError									:=	FALSE;			
// 			
// 		END_CASE

		bWeight1Actuator						:=	FALSE;
		bWeight2Actuator						:=	FALSE;		
		bWeight3Actuator						:=	FALSE;
		bWeight4Actuator						:=	FALSE;		

		IF NOT bError THEN
			udiErrorID										:= 0;
			sErrorDescription								:= '';
			sErrorDescription2								:= '';
			eState											:= E_Station.ePreparingToReady;
		ELSIF tonResetting.Q THEN                   	
			eState											:= E_Station.eError;
		END_IF
	//------------------------------------------------------------------------------
	E_Station.eManualMovement:     			// Stan ruchów manualnych  
	
		ACT_ManualMovements();
		//Wyjście z trybu serwisowego
		IF NOT bManualMovement THEN
			bWeight1Actuator								:=	bLastStateWeight1Actuator;
			bWeight2Actuator								:=	bLastStateWeight2Actuator;
			bWeight3Actuator								:=	bLastStateWeight3Actuator;
			bWeight4Actuator								:=	bLastStateWeight4Actuator;
			eState											:=	E_Station.eReady;
		END_IF
	//------------------------------------------------------------------------------
	
	E_Station.eHoming:						// Stan bazowania
	
		ACT_Homing();
		IF NOT bHoming AND tonHoming.Q THEN
			eState									:=	E_Station.ePreparingToReady;
		END_IF	
	//------------------------------------------------------------------------------
	
	E_Station.eHomingDone:                  // Stan wykonania bazowania
	
		bHomingDone											:= TRUE;		
		IF NOT bHoming THEN
			eState											:= E_Station.eReady;
		END_IF	
	//------------------------------------------------------------------------------
	
	
	E_Station.ePreparingToReady:            // Stan przygotowywania do gotowosci (zawsze przed Ready)
		//bHomingDone										:=	FALSE;	
		bWeight1Actuator									:=	FALSE;
		bWeight2Actuator									:=	FALSE;
		bWeight3Actuator									:=	FALSE;
		bWeight4Actuator									:=	FALSE;
		
		IF NOT bWasAborting THEN
			iFormsCounterWeight1								:= 3;	
			iFormsCounterWeight2								:= 2;
			iFormsCounterWeight3								:= 1;
			iFormsCounterWeight4								:= 0;
		END_IF
		
		IF tonPreparingToReadyDelay.Q THEN
			eState											:= E_Station.eReady;
		END_IF	
		
	//------------------------------------------------------------------------------
	
	
	E_Station.ePreparingToDisable:          // Stan przygotowywania do nieaktywnosci (po wyłączeniu Enable)	
		
		bWeight1Actuator									:=	FALSE;
		bWeight2Actuator									:=	FALSE;
		bWeight3Actuator									:=	FALSE;
		bWeight4Actuator									:=	FALSE;
		
		iFormsCounterWeight1								:= 3;	
		iFormsCounterWeight2								:= 2;
		iFormsCounterWeight3								:= 1;
		iFormsCounterWeight4								:= 0;
					
		eState												:= E_Station.eDisabled;
		eRunningState										:= E_WeightLiftStationState.eDisabled;
		
	//------------------------------------------------------------------------------
	
	
	E_Station.eReady:						// Stan gotowosci
		bWasAborting										:= FALSE;
		IF (bRun OR bAutoTare) AND bHomingDone AND NOT bCycleDone THEN
			eRunningState									:= E_WeightLiftStationState.eReady;
			eState											:= E_Station.eStarting;
		END_IF
		
		IF bHoming THEN
			eState											:= E_Station.eHoming;
		END_IF
		
		IF bManualMovement THEN
			bLastStateWeight1Actuator	:=	bManualWeight1Actuator	:=	bWeight1Actuator;
			bLastStateWeight2Actuator	:=	bManualWeight2Actuator	:=	bWeight2Actuator;
			bLastStateWeight3Actuator	:=	bManualWeight3Actuator	:=	bWeight3Actuator;
			bLastStateWeight4Actuator	:=	bManualWeight4Actuator	:=	bWeight4Actuator;		
			eState											:= E_Station.eManualMovement;
		END_IF
		
		IF NOT bRun THEN
			bCycleDone										:= FALSE;
		END_IF
		IF tonReadyAndRepair.Q THEN
			eRunningState									:= E_WeightLiftStationState.eReady;
		END_IF
	//------------------------------------------------------------------------------
	
	
	E_Station.eStopping:					// Stan zatrzymywania 

		ACT_Running();
		eState											:= E_Station.eReady;
		eRunningState									:= E_WeightLiftStationState.eReady;
		
		
	//------------------------------------------------------------------------------
	
	
	E_Station.eStarting:                  	// Stan uruchamiania (po Ready)
	
		eState												:= E_Station.eRunning;
	//------------------------------------------------------------------------------
	
	
	E_Station.eRunning:               		// Stan wykonywania cyklu (po Startingu), w tym stanie osobny
		
		ACT_Running();
		
		IF NOT bRun THEN
			eState											:= E_Station.eStopping;
		END_IF
		
		IF bCycleDone THEN
			eState											:= E_Station.eReady;
		END_IF
	//------------------------------------------------------------------------------
	
	
END_CASE
END_ACTION

ACTION ACT_ErrorHandling:
// Alarm_0300	300	Error	Podnoszenie wagi nr 1 | Blokada podnoszenia siłownika - sprawdź czujnik lub odblokuj
// Alarm_0301	301	Error	Podnoszenie wagi nr 2 | Blokada podnoszenia siłownika - sprawdź czujnik lub odblokuj
// Alarm_0302	302	Error	Podnoszenie wagi nr 3 | Blokada podnoszenia siłownika - sprawdź czujnik lub odblokuj
// Alarm_0303	303	Error	Podnoszenie wagi nr 4 | Blokada podnoszenia siłownika - sprawdź czujnik lub odblokuj
// Alarm_0304	304	Error	Podnoszenie wagi nr 5 | Blokada podnoszenia siłownika - sprawdź czujnik lub odblokuj
// Alarm_0305	305	Error	Podnoszenie wagi nr 6 | Blokada podnoszenia siłownika - sprawdź czujnik lub odblokuj

IF bAlarmInit THEN
    bAlarmInit := FALSE; 
	fbSourceInfo.Clear();
	fbSourceInfo.sName:=wsLiteral_TO_UTF8(sStationName);//'Machine';
	fbSourceInfo.nId:=udiStationIndex;//2700;
	// Alarm_0300	300	Error	Podnoszenie wagi nr 1 | Blokada podnoszenia siłownika - sprawdź czujnik lub odblokuj
    arfbAlarm[0].CreateEx(stEventEntry := TC_EVENTS.AlarmClass.Alarm_0300, bWithConfirmation:= FALSE,  ipSourceInfo:= fbSourceInfo); 
	// Alarm_0301	301	Error	Podnoszenie wagi nr 2 | Blokada podnoszenia siłownika - sprawdź czujnik lub odblokuj
	arfbAlarm[1].CreateEx(stEventEntry := TC_EVENTS.AlarmClass.Alarm_0301, bWithConfirmation:= FALSE,  ipSourceInfo:= fbSourceInfo);
	// Alarm_0302	302	Error	Podnoszenie wagi nr 3 | Blokada podnoszenia siłownika - sprawdź czujnik lub odblokuj
	arfbAlarm[2].CreateEx(stEventEntry := TC_EVENTS.AlarmClass.Alarm_0302, bWithConfirmation:= FALSE,  ipSourceInfo:= fbSourceInfo);
	// Alarm_0303	303	Error	Podnoszenie wagi nr 4 | Blokada podnoszenia siłownika - sprawdź czujnik lub odblokuj
	arfbAlarm[3].CreateEx(stEventEntry := TC_EVENTS.AlarmClass.Alarm_0303, bWithConfirmation:= FALSE,  ipSourceInfo:= fbSourceInfo);
	// Alarm_0304	304	Error	Podnoszenie wagi nr 5 | Blokada podnoszenia siłownika - sprawdź czujnik lub odblokuj
	arfbAlarm[4].CreateEx(stEventEntry := TC_EVENTS.AlarmClass.Alarm_0304, bWithConfirmation:= FALSE,  ipSourceInfo:= fbSourceInfo);
	// Alarm_0305	305	Error	Podnoszenie wagi nr 6 | Blokada podnoszenia siłownika - sprawdź czujnik lub odblokuj
	arfbAlarm[5].CreateEx(stEventEntry := TC_EVENTS.AlarmClass.Alarm_0305, bWithConfirmation:= FALSE,  ipSourceInfo:= fbSourceInfo);
END_IF

bStateError								:= (eState = E_Station.eError) OR (eState = E_Station.eResetting);

tonEventLogger (IN:= NOT tonEventLogger.Q, PT:=T#1S);

IF tonEventLogger.Q THEN
	
	// Alarm_0300	300	Error	Podnoszenie wagi nr 1 | Blokada podnoszenia siłownika - sprawdź czujnik lub odblokuj
	// Alarm_0304	304	Error	Podnoszenie wagi nr 5 | Blokada podnoszenia siłownika - sprawdź czujnik lub odblokuj
	//Błąd podnoszenia wagi 1 
	tonWeight1ActuatorUpError				(IN:= bWeight1Actuator AND NOT bWeight1ActuatorSensorUp	, PT:=T#2S);
	IF tonWeight1ActuatorUpError.Q THEN
		IF NOT bTwoPhaseMode AND NOT arfbAlarm[0].bActive THEN
			arfbAlarm[0].Raise(nTimeStamp:=0);
		END_IF
		IF bTwoPhaseMode AND NOT arfbAlarm[4].bActive THEN
				arfbAlarm[4].Raise(nTimeStamp:=0);
		END_IF
		IF (arfbAlarm[0].bActive OR arfbAlarm[4].bActive) AND bReset THEN
			bWeight1Actuator			:= FALSE;
		END_IF
		ELSE	
		IF NOT bTwoPhaseMode AND arfbAlarm[0].bActive AND bReset THEN
			arfbAlarm[0].Clear(nTimeStamp:=0, bResetConfirmation:= FALSE);
		END_IF
		IF bTwoPhaseMode AND arfbAlarm[4].bActive AND bReset THEN
			arfbAlarm[4].Clear(nTimeStamp:=0, bResetConfirmation:= FALSE);
		END_IF
	// 	bError								:= TRUE;
	// 	IF NOT bTwoPhaseMode THEN
	// 	udiErrorID							:= 191;	
	// 	//udiErrorID 						:= udiErrorID + udiStationIndex;
	// 	sErrorDescription					:= 'Podnoszenie wagi nr 1';
	// 	END_IF
	// 	
	// 	IF bTwoPhaseMode THEN
	// 		udiErrorID						:= 195;
	// 		sErrorDescription				:= 'Podnoszenie wagi nr 5';
	// 	END_IF
	// 	sErrorDescription2					:= 'Blokada podnoszenia siłownika - sprawdź czujnik lub odblokuj';
	END_IF
	// Alarm_0301	301	Error	Podnoszenie wagi nr 2 | Blokada podnoszenia siłownika - sprawdź czujnik lub odblokuj
	// Alarm_0305	305	Error	Podnoszenie wagi nr 6 | Blokada podnoszenia siłownika - sprawdź czujnik lub odblokuj
	//Błąd podnoszenia wagi 2
	tonWeight2ActuatorUpError				(IN:= bWeight2Actuator AND NOT bWeight2ActuatorSensorUp	, PT:=T#2S);
	IF tonWeight2ActuatorUpError.Q THEN
		
		IF NOT bTwoPhaseMode AND NOT arfbAlarm[1].bActive THEN
				arfbAlarm[1].Raise(nTimeStamp:=0);
		END_IF
		IF bTwoPhaseMode AND NOT arfbAlarm[5].bActive THEN
				arfbAlarm[5].Raise(nTimeStamp:=0);
		END_IF	
		IF (arfbAlarm[1].bActive OR arfbAlarm[5].bActive) AND bReset THEN
			bWeight1Actuator			:= FALSE;
		END_IF
		ELSE	
		IF NOT bTwoPhaseMode AND arfbAlarm[1].bActive AND bReset THEN
			arfbAlarm[1].Clear(nTimeStamp:=0, bResetConfirmation:= FALSE);
		END_IF	
		IF bTwoPhaseMode AND arfbAlarm[5].bActive AND bReset THEN
			arfbAlarm[5].Clear(nTimeStamp:=0, bResetConfirmation:= FALSE);
		END_IF	
	// 	bError								:= TRUE;
	// 	IF NOT bTwoPhaseMode THEN
	// 	udiErrorID							:= 192;	
	// 	//udiErrorID 						:= udiErrorID + udiStationIndex;
	// 	sErrorDescription					:= 'Podnoszenie wagi nr 2';
	// 	END_IF
	
	// 	IF bTwoPhaseMode THEN
	// 		udiErrorID						:= 196;
	// 		sErrorDescription				:= 'Podnoszenie wagi nr 6';
	// 	END_IF
	// 	sErrorDescription2					:= 'Blokada podnoszenia siłownika - sprawdź czujnik lub odblokuj';	
	END_IF
	// Alarm_0302	302	Error	Podnoszenie wagi nr 3 | Blokada podnoszenia siłownika - sprawdź czujnik lub odblokuj
	//Błąd podnoszenia wagi 3
	tonWeight3ActuatorUpError				(IN:= bWeight3Actuator AND NOT bWeight3ActuatorSensorUp	OR bTest, PT:=T#2S);
	IF tonWeight3ActuatorUpError.Q THEN
		IF NOT arfbAlarm[2].bActive THEN
				arfbAlarm[2].Raise(nTimeStamp:=0);
			END_IF
		ELSE	
			IF  arfbAlarm[2].bActive AND bReset THEN
				arfbAlarm[2].Clear(nTimeStamp:=0, bResetConfirmation:= FALSE);
			END_IF	
	// 	bError								:= TRUE;
	// 	udiErrorID							:= 193;	
	// 	//udiErrorID 						:= udiErrorID + udiStationIndex;
	// 	sErrorDescription					:= 'Podnoszenie wagi nr 3';
	// 	sErrorDescription2					:= 'Blokada podnoszenia siłownika - sprawdź czujnik lub odblokuj';
	END_IF
	// Alarm_0303	303	Error	Podnoszenie wagi nr 4 | Blokada podnoszenia siłownika - sprawdź czujnik lub odblokuj
	//Błąd podnoszenia wagi 4
	tonWeight4ActuatorUpError				(IN:= bWeight4Actuator AND NOT bWeight4ActuatorSensorUp	, PT:=T#2S);
	IF tonWeight4ActuatorUpError.Q THEN
		IF NOT arfbAlarm[3].bActive THEN
				arfbAlarm[3].Raise(nTimeStamp:=0);
			END_IF
		ELSE	
			IF  arfbAlarm[3].bActive AND bReset THEN
				arfbAlarm[3].Clear(nTimeStamp:=0, bResetConfirmation:= FALSE);
			END_IF	
	// 	bError								:= TRUE;
	// 	udiErrorID							:= 194;	
	// 	//udiErrorID 						:= udiErrorID + udiStationIndex;
	// 	sErrorDescription					:= 'Podnoszenie wagi nr 4';
	// 	sErrorDescription2					:= 'Blokada podnoszenia siłownika - sprawdź czujnik lub odblokuj';
	END_IF
	
	IF NOT bEnable OR NOT bEStop THEN
		bError								:= FALSE;
	END_IF
	
	IF bError AND NOT bStateError THEN
		eState								:= E_Station.eError;
	END_IF
	
	(*Przepisywanie nazwy stacji*)
	sErrorStationName						:= WSTRING_TO_STRING(sStationName);
	
	(*Wyświetlanie błedu na wyjściu*)
	bError									:= FALSE;
	
	FOR nAlarmNumerator := 0 TO 19 DO
		bError								:= bError OR arfbAlarm[nAlarmNumerator].bActive;
	END_FOR
END_IF
END_ACTION

ACTION ACT_Homing:
bWeight1Actuator						:= FALSE;
bWeight2Actuator						:= FALSE;
bWeight3Actuator						:= FALSE;
bWeight4Actuator						:= FALSE;

iFormsCounterWeight1					:= 0;
iFormsCounterWeight2					:= 1;
iFormsCounterWeight3					:= 2;
iFormsCounterWeight4					:= 3;

eState									:= E_Station.eHomingDone;
END_ACTION

ACTION ACT_ManualMovements:


IF NOT bRun (*AND bManualMovement*) THEN
	
	bWeight1Actuator		:=	bManualWeight1Actuator;
	bWeight2Actuator		:=	bManualWeight2Actuator;
	bWeight3Actuator		:=	bManualWeight3Actuator;
	bWeight4Actuator		:=	bManualWeight4Actuator;	
ELSE
	bManualWeight1Actuator	:=	FALSE;
	bManualWeight2Actuator	:=	FALSE;
	bManualWeight3Actuator	:=	FALSE;
	bManualWeight4Actuator	:=	FALSE;		
END_IF


IF bHoming THEN
	eState											:= E_Station.eHoming;
END_IF

//Running();

IF NOT bRun THEN
	bCycleDone 										:= FALSE;
END_IF
END_ACTION

ACTION ACT_Running:

CASE eRunningState OF
	
	E_WeightLiftStationState.eRepair:		//Naprawa
		
		bWeight1Actuator								:= FALSE;
		bWeight2Actuator								:= FALSE;
		bWeight3Actuator								:= FALSE;
		bWeight4Actuator								:= FALSE;
		
		iFormsCounterWeight4							:= 0;	
		iFormsCounterWeight3							:= 1;
		iFormsCounterWeight2							:= 2;
		iFormsCounterWeight1							:= 3;
		
		IF bTwoPhaseMode THEN
			iFormsCounterWeight2						:= 0;
			iFormsCounterWeight1						:= 1;
		END_IF
		
		IF NOT arrWeightPackageState[1].bFormPresent AND NOT arrWeightPackageState[2].bFormPresent AND NOT arrWeightPackageState[3].bFormPresent AND NOT arrWeightPackageState[4].bFormPresent THEN
			
			IF tonRepairOnDelay.Q THEN
				eRunningState							:= E_WeightLiftStationState.ePrepareToStorageOfForms;	
			END_IF
	
		END_IF
		

	E_WeightLiftStationState.eDisabled :	//Stan wyłączony
	
		eRunningState									:= E_WeightLiftStationState.eReady;
		
	//----------------------------------------------------------------------------------------
		
	E_WeightLiftStationState.eReady :		//Sprawdzam co się dzieje ze stacją
	
(*	w1
		//IF bDeparture THEN
			
			//eRunningState								:= E_WeightLiftStationState.ePrepareToStorageOfForms;
			
		IF NOT bWeight1FormSensor AND NOT bWeight2FormSensor AND NOT bWeight3FormSensor AND NOT bWeight4FormSensor THEN //Nie ma wszystkich formatek
		
			iFormsCounterWeight4						:= 0;	
			iFormsCounterWeight3						:= 1;
			iFormsCounterWeight2						:= 2;
			iFormsCounterWeight1						:= 3;
			eRunningState								:= E_WeightLiftStationState.ePrepareToStorageOfForms;

		//Przechodzę do opuszczanie formatek
		ELSIF bWeight1FormSensor AND bWeight2FormSensor AND bWeight3FormSensor AND bWeight4FormSensor THEN //Mamy wszystkie formateki
			
			iFormsCounterWeight4						:= 0;	
			iFormsCounterWeight3						:= 0;
			iFormsCounterWeight2						:= 0;
			iFormsCounterWeight1						:= 0;
			eRunningState								:= E_WeightLiftStationState.eWeighingCycleON;	
			
		ELSE
			//eRunningState								:= E_WeightLiftStationState.eRepair;
			eRunningState								:= E_WeightLiftStationState.ePrepareToStorageOfForms;			
		END_IF
*)		

	(*	w2	*)
		
		IF NOT bAutoTare THEN
			eRunningState								:= E_WeightLiftStationState.ePrepareToStorageOfForms;		
		ELSE
			CASE iCaseTareWeights OF
				0:
					iCaseTareWeights	:=	iCaseTareWeights	+	10;
				10:
				 IF tonWeightsEmpty.Q THEN
					 iCaseTareWeights	:=	iCaseTareWeights	+	10;
				 END_IF
				20:
					bWeight1Actuator	:= TRUE;
					bWeight2Actuator	:= TRUE;
					bWeight3Actuator	:= NOT bTwoPhaseMode;
					bWeight4Actuator	:= NOT bTwoPhaseMode;				
					iCaseTareWeights	:= iCaseTareWeights	+	10;
				30:
					IF toniCaseTareWeights1.Q THEN
						iCaseTareWeights:=	iCaseTareWeights	+	10;
					END_IF
				40:
					bTareWeights		:= TRUE;
					iCaseTareWeights	:= iCaseTareWeights	+	10;	
				50:
					IF toniCaseTareWeights2.Q THEN
						bAutoTare		:= FALSE;
						bTareWeights	:= FALSE;
						iCaseTareWeights:= 0;
					END_IF				
			END_CASE
		END_IF
		
		
		
	//----------------------------------------------------------------------------------------	

	E_WeightLiftStationState.ePrepareToStorageOfForms: //Przygotowywanie do magazynowania formatek
		
		bWeight1Actuator								:= FALSE;
		bWeight2Actuator								:= FALSE;
		bWeight3Actuator								:= FALSE;
		bWeight4Actuator								:= FALSE;
		
		eRunningState									:=  E_WeightLiftStationState.eStorageOfForms;	
	//----------------------------------------------------------------------------------------		
	
	E_WeightLiftStationState.eStorageOfForms:	//Magazynuje formatki
		
		//Waga 1/5====================================================================================================================
		IF (tonWeight1ActuatorDelay.Q OR bCountingBeforeSensorsMode) AND ((	iFormsCounterWeight1 = 4 AND NOT	bTwoPhaseMode) OR 
																			iFormsCounterWeight1 = 2 AND 		bTwoPhaseMode) THEN	
			bWeight1Actuator	:= TRUE;
		END_IF
		
		//Waga 2/6=====================================================================================================================		
		IF (tonWeight2ActuatorDelay.Q OR bCountingBeforeSensorsMode) AND ((	iFormsCounterWeight2 = 4  AND NOT	bTwoPhaseMode) OR 
																			iFormsCounterWeight2 = 2 AND 		bTwoPhaseMode) THEN	
			bWeight2Actuator	:= TRUE;
		END_IF
		
		//Waga 3====================================================================================================================
		IF (tonWeight3ActuatorDelay.Q OR bCountingBeforeSensorsMode) AND iFormsCounterWeight3 = 4	THEN //Podnoszenie Waga 3
			bWeight3Actuator	:= NOT bTwoPhaseMode;
		END_IF
			
		//Waga 4=====================================================================================================================	
		IF (tonWeight4ActuatorDelay.Q OR bCountingBeforeSensorsMode) AND iFormsCounterWeight4 = 4	THEN //Podnoszenie Waga 4
			bWeight4Actuator	:= NOT bTwoPhaseMode;
		END_IF

		
		IF (bWeight1ActuatorSensorUp) AND (bWeight2ActuatorSensorUp) AND
 		   (bWeight3ActuatorSensorUp OR bTwoPhaseMode) AND (bWeight4ActuatorSensorUp OR bTwoPhaseMode) THEN
		   		eRunningState								:= E_WeightLiftStationState.eWeighingCycleStart;
		   
		END_IF
		
	//----------------------------------------------------------------------------------------
	
	E_WeightLiftStationState.eWeighingCycleStart:	//Rozpoczęcie Ważenia
	
		IF bWeighingCycle THEN
			eRunningState								:= E_WeightLiftStationState.eWeighingCycleON;
		END_IF

	//----------------------------------------------------------------------------------------

	
	E_WeightLiftStationState.eWeighingCycleON:	//Trwa ważenie
	
		IF (arrWeightPackageState[1].bWeighed OR arrWeightPackageState[1].bWeightAborted) AND (arrWeightPackageState[2].bWeighed OR arrWeightPackageState[2].bWeightAborted) AND
		   (arrWeightPackageState[3].bWeighed OR arrWeightPackageState[3].bWeightAborted OR bTwoPhaseMode) AND (arrWeightPackageState[4].bWeighed OR arrWeightPackageState[4].bWeightAborted OR bTwoPhaseMode) THEN  //Czekam na przepisanie statusów z wag
		   bWeighingCycleDone	:=	TRUE;
			IF bCanReleaseForms THEN			//Mogę wypuścić formatki
				eRunningState							:= E_WeightLiftStationState.eWeightLiftDown;
				bWeighingCycleDone	:=	FALSE;
			END_IF
			
		END_IF
	//----------------------------------------------------------------------------------------
	
	
	E_WeightLiftStationState.eWeightLiftDown:	//Opuszczanie formatek
		
		bWeight1Actuator								:= FALSE;
		bWeight2Actuator								:= FALSE;
		bWeight3Actuator								:= FALSE;
		bWeight4Actuator								:= FALSE;
		
		iFormsCounterWeight4							:= 0;	
		iFormsCounterWeight3							:= 0;
		iFormsCounterWeight2							:= 0;
		iFormsCounterWeight1							:= 0;
		
		IF tonWeightAntuatorOffDelay.Q THEN	        
			eRunningState								:= E_WeightLiftStationState.eDepartureOfForms;
		END_IF	
	//----------------------------------------------------------------------------------------
	
	E_WeightLiftStationState.eDepartureOfForms:	//Wypuszczamy formatki

			eRunningState								:= E_WeightLiftStationState.eDone;
			bDeparture									:= TRUE;

	//----------------------------------------------------------------------------------------
	
	E_WeightLiftStationState.eDone:				//Cykl skończony
		
			bCycleDone									:= TRUE;		//Wystawiam koniec cyklu
			eRunningState								:= E_WeightLiftStationState.eReady;
		
			
END_CASE
END_ACTION

ACTION ACT_Signals:
//TONs
tonWeight1ActuatorDelay		(IN:= eRunningState = E_WeightLiftStationState.eStorageOfForms AND bWeight1FormSensor, PT:= tWeight1ActuatorUpDelay);
tonWeight2ActuatorDelay		(IN:= eRunningState = E_WeightLiftStationState.eStorageOfForms AND bWeight2FormSensor, PT:= tWeight2ActuatorUpDelay);
tonWeight3ActuatorDelay		(IN:= eRunningState = E_WeightLiftStationState.eStorageOfForms AND bWeight3FormSensor, PT:= tWeight3ActuatorUpDelay);
tonWeight4ActuatorDelay		(IN:= eRunningState = E_WeightLiftStationState.eStorageOfForms AND bWeight4FormSensor, PT:= tWeight4ActuatorUpDelay);
tonWeightAntuatorOffDelay 	(IN:= NOT bWeight1Actuator AND NOT bWeight2Actuator AND NOT bWeight3Actuator AND NOT bWeight4Actuator, PT:=T#100MS);

tonPreparingToReadyDelay	(IN:= eState = E_Station.ePreparingToReady			,PT:= T#300MS);
tonResetting				(IN:= eState = E_Station.eResetting					,PT:= T#200MS);
tonHoming					(IN:= eState = E_Station.eHoming					,PT:= T#1S);
rtResetCommands				(CLK:=eState = E_Station.eReady 					,Q=>); 
tonReadyAndRepair			(IN:= eState = E_Station.eReady AND eRunningState = E_WeightLiftStationState.eRepair, PT:=T#10S);
//Triggers

rtWeight1FormSensor			(CLK:= bWeight1FormSensor AND NOT bCountingBeforeSensorsMode);
rtWeight2FormSensor			(CLK:= bWeight2FormSensor AND NOT bCountingBeforeSensorsMode);
rtWeight3FormSensor			(CLK:= bWeight3FormSensor AND NOT bCountingBeforeSensorsMode);
rtWeight4FormSensor			(CLK:= bWeight4FormSensor AND NOT bCountingBeforeSensorsMode);

ftWeight1FormBeforeSensor	(CLK:=bWeight1FormBeforeSensor AND bCountingBeforeSensorsMode AND NOT bWeight1ActuatorSensorUp, Q=>);
ftWeight2FormBeforeSensor	(CLK:=bWeight2FormBeforeSensor AND bCountingBeforeSensorsMode AND NOT bWeight2ActuatorSensorUp, Q=>);
ftWeight3FormBeforeSensor	(CLK:=bWeight3FormBeforeSensor AND bCountingBeforeSensorsMode AND NOT bWeight3ActuatorSensorUp, Q=>);
ftWeight4FormBeforeSensor	(CLK:=bWeight4FormBeforeSensor AND bCountingBeforeSensorsMode AND NOT bWeight4ActuatorSensorUp, Q=>);

//
tonWeightsEmpty			(IN:= iCaseTareWeights = 10 AND NOT bWeight1FormSensor AND NOT bWeight2FormSensor AND NOT bWeight3FormSensor AND NOT bWeight4FormSensor, PT:=T#3S);	
toniCaseTareWeights1	(IN:= iCaseTareWeights = 30, PT:= T#3S);	
toniCaseTareWeights2	(IN:= iCaseTareWeights = 50, PT:= T#3S);	

//=========================================================================================================================================================

//Licznik formatek w górę
tofRunning(IN:= eState = E_Station.eRunning OR eState = E_Station.eStopping OR  eGlobalState=E_PMLState.ePMLState_STOPPING OR eGlobalState=E_PMLState.ePMLState_EXECUTE OR eGlobalState=E_PMLState.ePMLState_STARTING, PT:=T#3S);
//IF eState = E_Station.eRunning OR eState = E_Station.eStopping OR  (eGlobalState=E_PMLState.ePMLState_STOPPING OR eGlobalState=E_PMLState.ePMLState_EXECUTE OR eGlobalState=E_PMLState.ePMLState_STARTING) THEN 
IF tofRunning.Q THEN

	//Liczymy Formatki na Wadze 1 
	IF rtWeight1FormSensor.Q OR ftWeight1FormBeforeSensor.Q THEN
		iFormsCounterWeight1								:= iFormsCounterWeight1 + 1;
	END_IF
	
	//Liczymy Formatki na Wadze 2 
	IF rtWeight2FormSensor.Q OR ftWeight2FormBeforeSensor.Q THEN
		iFormsCounterWeight2								:= iFormsCounterWeight2 + 1;
	END_IF

	//Liczymy Formatki na Wadze 3 
	IF rtWeight3FormSensor.Q OR ftWeight3FormBeforeSensor.Q THEN
		iFormsCounterWeight3								:= iFormsCounterWeight3 + 1;
	END_IF
	
	//Liczymy Formatki na Wadze 4 
	IF rtWeight4FormSensor.Q OR ftWeight4FormBeforeSensor.Q THEN
		iFormsCounterWeight4								:= iFormsCounterWeight4 + 1;
	END_IF

END_IF

//=========================================================================================================================================================
END_ACTION

ACTION ACT_Statistics:

//Statystyka do zliczania czasu cyklu 
rtrigCycleTimerRead(CLK:=bCycleDone);

	IF rtrigCycleTimerRead.Q THEN
		tCycleTime:=tonCycleTimer.ET;
		tt:=tt+1;
	END_IF
	
tonCycleTimer(IN:= eRunningState>E_WeightLiftStationState.eReady , PT:=T#1D);
END_ACTION

ACTION aRepair:
tonRepairOnDelay			(IN:= eState = E_Station.eRunning AND eRunningState = E_WeightLiftStationState.eRepair AND bRepairAllRegistersAreEmpty, PT:= T#2S);

bRepairAllRegistersAreEmpty	:= (NOT arrWeightPackageState[1].bFormPresent AND NOT arrWeightPackageState[2].bFormPresent AND NOT arrWeightPackageState[3].bFormPresent AND NOT arrWeightPackageState[4].bFormPresent);// AND


(** 1 **********************************************************************************************)
tonRepair1(IN:=
									eRunningState = E_WeightLiftStationState.eWeighingCycleON AND
									eState = E_Station.eRunning AND
									bCanReleaseForms AND 
									bConveyorRunning AND 				
									(
									NOT arrWeightPackageState[1].bWeighed OR
									NOT arrWeightPackageState[2].bWeighed OR 
		  							NOT arrWeightPackageState[3].bWeighed OR  
									NOT arrWeightPackageState[4].bWeighed	
									) AND 
									bWeight1FormSensor AND 
									bWeight2FormSensor AND 
									bWeight3FormSensor AND 									
									bWeight4FormSensor 	AND
									NOT tonRepair1.Q							
							, PT:=T#10S);
							
IF 	tonRepair1.Q THEN
	eRunningState		:= E_WeightLiftStationState.eRepair;
	iRepair1 			:= iRepair1	+	1;
END_IF					
(****************************************************************************************************)
(** 2 **********************************************************************************************)
tonRepair2(IN:=
									eRunningState = E_WeightLiftStationState.eStorageOfForms AND
									eState = E_Station.eRunning AND
									bCanReleaseForms AND
									bConveyorRunning AND 
									//(
									//NOT arrWeightPackageState[1].bWeighed OR
									////NOT arrWeightPackageState[2].bWeighed OR 
		  							//NOT arrWeightPackageState[3].bWeighed OR  
									//NOT arrWeightPackageState[4].bWeighed	
									//) AND 
									(
									bWeight1FormSensor OR
									bWeight2FormSensor OR 
									bWeight3FormSensor OR 									
									bWeight4FormSensor 
									) AND
									NOT tonRepair2.Q							
							, PT:=T#10S);
							
IF 	tonRepair2.Q THEN
	eRunningState		:= E_WeightLiftStationState.eRepair;
	iRepair2 			:= iRepair2	+	1;
END_IF					
(****************************************************************************************************)
(** 3 **********************************************************************************************)
tonRepair3(IN:=
									eRunningState = E_WeightLiftStationState.eWeighingCycleON AND
									eState = E_Station.eRunning AND
									bCanReleaseForms AND 
									bConveyorRunning AND 
									(
									NOT arrWeightPackageState[1].bWeighed OR
									NOT arrWeightPackageState[2].bWeighed OR 
		  							NOT arrWeightPackageState[3].bWeighed OR  
									NOT arrWeightPackageState[4].bWeighed	
									) AND 
									NOT bWeight1FormSensor AND 
									NOT bWeight2FormSensor AND 
									NOT bWeight3FormSensor AND 									
									NOT bWeight4FormSensor AND
									NOT tonRepair3.Q							
							, PT:=T#10S);
							
IF 	tonRepair3.Q THEN
	eRunningState		:= E_WeightLiftStationState.eRepair;
	iRepair3 			:= iRepair3	+	1;
END_IF					
(****************************************************************************************************)
(** 4 **********************************************************************************************)
tonRepair4(IN:=
									
									eState = E_Station.eRunning AND
									bCanReleaseForms AND 
									bConveyorRunning AND 
									(
									iFormsCounterWeight1 > 4 OR
									iFormsCounterWeight2 > 4 OR
		  							iFormsCounterWeight3 > 4 OR   
									iFormsCounterWeight4 > 4 
									) AND 
									NOT bWeight1FormSensor AND 
									NOT bWeight2FormSensor AND 
									NOT bWeight3FormSensor AND 									
									NOT bWeight4FormSensor AND
									NOT tonRepair4.Q							
							, PT:=T#10S);
							
IF 	tonRepair4.Q THEN
	eRunningState		:= E_WeightLiftStationState.eRepair;
	iRepair4 			:= iRepair4	+	1;
END_IF					
(****************************************************************************************************)

(** 5 **********************************************************************************************)
tonRepair5(IN:=
									
									eState = E_Station.eRunning AND
									bCanReleaseForms AND
									bConveyorRunning AND 									
									bTwoPhaseMode AND 
									(
									iFormsCounterWeight1 > 2 OR
									iFormsCounterWeight2 > 2 
									) AND 
									//NOT bWeight1FormSensor AND 
									//NOT bWeight2FormSensor AND 

									NOT tonRepair5.Q							
							, PT:=T#8S);
							
IF 	tonRepair5.Q THEN
	eRunningState		:= E_WeightLiftStationState.eRepair;
	iRepair5 			:= iRepair5	+	1;
END_IF					
(****************************************************************************************************)

(** 6 **********************************************************************************************)
tonRepair6(IN:=
									
									(eState = E_Station.eReady OR (eState = E_Station.eRunning AND eRunningState=E_WeightLiftStationState.eStorageOfForms))
									AND
									bCanReleaseForms AND
									bConveyorRunning AND 									
									
									(
									bWeight1Actuator OR
									bWeight2Actuator OR
									bWeight3Actuator OR									
									bWeight4Actuator 								
									) AND 
									NOT tonRepair6.Q							
							, PT:=T#8S);
							
IF 	tonRepair6.Q THEN
	eRunningState			:= E_WeightLiftStationState.eRepair;
	bWeight1Actuator		:= FALSE;
	bWeight2Actuator		:= FALSE;
	bWeight3Actuator		:= FALSE;
	bWeight4Actuator		:= FALSE;	
	iFormsCounterWeight4	:= 0;	
	iFormsCounterWeight3	:= 1;
	iFormsCounterWeight2	:= 2;
	iFormsCounterWeight1	:= 3;	
	iRepair6 				:= iRepair6	+	1;
END_IF					
(****************************************************************************************************)
END_ACTION

ACTION aResetCommands:



bManualWeight1Actuator	:=	FALSE;
bManualWeight2Actuator	:=	FALSE;
bManualWeight3Actuator	:=	FALSE;
bManualWeight4Actuator	:=	FALSE;

bLastStateWeight1Actuator:=	FALSE;
bLastStateWeight2Actuator:=	FALSE;
bLastStateWeight3Actuator:=	FALSE;
bLastStateWeight4Actuator:=	FALSE;

bWeight1Actuator	:=	FALSE;
bWeight2Actuator	:=	FALSE;
bWeight3Actuator	:=	FALSE;
bWeight4Actuator	:=	FALSE;
		

iFormsCounterWeight4	:= 0;	
iFormsCounterWeight3	:= 1;
iFormsCounterWeight2	:= 2;
iFormsCounterWeight1	:= 3;
IF bTwoPhaseMode THEN
	iFormsCounterWeight2	:= 0;
	iFormsCounterWeight1	:= 1;
END_IF


bResetCycleOn			:=	FALSE;	
bWeighingCycleDone		:=	FALSE;
END_ACTION

ACTION aResetCommandsAborting:



bManualWeight1Actuator	:=	FALSE;
bManualWeight2Actuator	:=	FALSE;
bManualWeight3Actuator	:=	FALSE;
bManualWeight4Actuator	:=	FALSE;

bLastStateWeight1Actuator:=	FALSE;
bLastStateWeight2Actuator:=	FALSE;
bLastStateWeight3Actuator:=	FALSE;
bLastStateWeight4Actuator:=	FALSE;

bWeight1Actuator	:=	FALSE;
bWeight2Actuator	:=	FALSE;
bWeight3Actuator	:=	FALSE;
bWeight4Actuator	:=	FALSE;
		

(*iFormsCounterWeight4	:= 0;	
iFormsCounterWeight3	:= 1;
iFormsCounterWeight2	:= 2;
iFormsCounterWeight1	:= 3;
IF bTwoPhaseMode THEN
	iFormsCounterWeight2	:= 0;
	iFormsCounterWeight1	:= 1;
END_IF*)


bResetCycleOn			:=	FALSE;	
bWeighingCycleDone		:=	FALSE;
END_ACTION

ACTION aStationID:
udiStationID	:=	udiStationIndex;
END_ACTION

ACTION ResetAll:
(*****Reset bloczka*****)
IF bEnable THEN
	IF eState <> E_Station.eDisabled AND eState <> E_Station.ePreparingToDisable THEN
		IF bResetCycle THEN
			bResetCycleOn						:= TRUE;
			eState								:= E_Station.ePreparingToReady;
		END_IF
	END_IF
END_IF


IF bResetCycleOn THEN
	
	aResetCommands();
	eRunningState							:= E_WeightLiftStationState.eReady;	
	eState 				 					:= E_Station.eReady;

END_IF
END_ACTION

END_FUNCTION_BLOCK

// ---- POUs/FB/Charts/FB_WeightHistory.TcPOU
FUNCTION_BLOCK FB_WeightHistory
VAR_INPUT
    eWeight1RunningState : INT;
    eWeight2RunningState : INT;
    eWeight3RunningState : INT;
    eWeight4RunningState : INT;

    WeightMeasured_1      : LREAL;
    CorrectionWeight_1    : LREAL;
    WeightMeasured_2      : LREAL;
    CorrectionWeight_2    : LREAL;
    WeightMeasured_3      : LREAL;
    CorrectionWeight_3    : LREAL;
    WeightMeasured_4      : LREAL;
    CorrectionWeight_4    : LREAL;
END_VAR

VAR_IN_OUT
    aWeightPoints : ARRAY [0..7,0..9999] OF ST_Point_1;
END_VAR

VAR
    fbTrig1 : R_TRIG;
    fbTrig2 : R_TRIG;
    fbTrig3 : R_TRIG;
    fbTrig4 : R_TRIG;

	fileTime : T_FILETIME64;
    dtNow    : DT;

    i           : INT;
END_VAR

// ----------------------------------------
// 1) Pobierz aktualny czas systemowy (FILETIME64)
// ----------------------------------------
fileTime := F_GetSystemTime();

// ----------------------------------------
// 2) FILETIME64 → DT (pełna data i czas)
// ----------------------------------------
dtNow := FILETIME64_TO_DT(fileTime);




// --------------------------	
// WAGA 1
// --------------------------
fbTrig1(CLK := (eWeight1RunningState = 3));   // flanka na stanie 3
IF fbTrig1.Q THEN
    // kolumna 0: WeightMeasured
    FOR i := 0 TO 9998 DO
        aWeightPoints[0, i] := aWeightPoints[0, i + 1];
    END_FOR
    aWeightPoints[0, 9999].x := dtNow;
    aWeightPoints[0, 9999].y := LREAL_TO_INT(WeightMeasured_1);

    // kolumna 1: CorrectionWeight
    FOR i := 0 TO 9998 DO
        aWeightPoints[4, i] := aWeightPoints[4, i + 1];
    END_FOR
    aWeightPoints[4, 9999].x := dtNow;
    aWeightPoints[4, 9999].y := LREAL_TO_INT(CorrectionWeight_1);
END_IF


// --------------------------
// WAGA 2
// --------------------------
fbTrig2(CLK := (eWeight2RunningState = 3));
IF fbTrig2.Q THEN
    // kolumna 2: WeightMeasured
    FOR i := 0 TO 9998 DO
        aWeightPoints[1, i] := aWeightPoints[1, i + 1];
    END_FOR
    aWeightPoints[1, 9999].x := dtNow;
    aWeightPoints[1, 9999].y := LREAL_TO_INT(WeightMeasured_2);

    // kolumna 3: CorrectionWeight
    FOR i := 0 TO 9998 DO
        aWeightPoints[5, i] := aWeightPoints[5, i + 1];
    END_FOR
    aWeightPoints[5, 9999].x := dtNow;
    aWeightPoints[5, 9999].y := LREAL_TO_INT(CorrectionWeight_2);
END_IF


// --------------------------
// WAGA 3
// --------------------------
fbTrig3(CLK := (eWeight3RunningState = 3));
IF fbTrig3.Q THEN
    // kolumna 4: WeightMeasured
    FOR i := 0 TO 9998 DO
        aWeightPoints[2, i] := aWeightPoints[2, i + 1];
    END_FOR
    aWeightPoints[2, 9999].x := dtNow;
    aWeightPoints[2, 9999].y := LREAL_TO_INT(WeightMeasured_3);

    // kolumna 5: CorrectionWeight
    FOR i := 0 TO 9998 DO
        aWeightPoints[6, i] := aWeightPoints[6, i + 1];
    END_FOR
    aWeightPoints[6, 9999].x := dtNow;
    aWeightPoints[6, 9999].y := LREAL_TO_INT(CorrectionWeight_3);
END_IF


// --------------------------
// WAGA 4
// --------------------------
// UWAGA: tu według Twojego opisu stan = 4
fbTrig4(CLK := (eWeight4RunningState = 3));
IF fbTrig4.Q THEN
    // kolumna 6: WeightMeasured
    FOR i := 0 TO 9998 DO
        aWeightPoints[3, i] := aWeightPoints[3, i + 1];
    END_FOR
    aWeightPoints[3, 9999].x := dtNow;
    aWeightPoints[3, 9999].y := LREAL_TO_INT(WeightMeasured_4);

    // kolumna 7: CorrectionWeight
    FOR i := 0 TO 9998 DO
        aWeightPoints[7, i] := aWeightPoints[7, i + 1];
    END_FOR
    aWeightPoints[7, 9999].x := dtNow;
    aWeightPoints[7, 9999].y := LREAL_TO_INT(CorrectionWeight_4);
END_IF

END_FUNCTION_BLOCK

// ---- POUs/P11_CapCorrectCheck.TcPOU
PROGRAM P11_CapCorrectCheck
VAR_INPUT
	IbCapCorrectCheckCapOKSensor 			AT %I*	: BOOL;			// Wejście wykrycia nasadki 
	IbCapCorrectCheckCapNotScrewedSensor 	AT %I*	: BOOL;			// Wejście wykrycia złego zakręcenia 
	IbCapCorrectCheckBottleSensor 			AT %I*	: BOOL;			// Wejście wykrycia butelki	
	IbCapCorrectCheckAfterScrewerFormSensor AT %I*	: BOOL;			// Wejście wykrycia formatek w sprawdzaniu nasade
	IbCapCorrectCheckFormSensor 			AT %I*	: BOOL;			// Wejście wykrycia formatek w sprawdzaniu nasade
	IbCapCorrectCheckDialAfterScrewerFormSensor AT %I*	: BOOL;			// Wejście wykrycia formatek na skos
END_VAR
VAR
	fbCapCorrectCheck					:FB_Checker;
	eCapCorrectCheckState				:E_Station; 			// Stan pracy sprawdzanie zakrecenia			
	eCapCorrectCheckRunningState		:E_CheckerState; 		// Stan pracy sprawdzania zakrecenie
	fbCapCorrectCheckState				:FB_State;
	
	IbCapCorrectCheckHeightEncoderPulses 	AT %I*: BOOL;			// Enkoder podnośnika czujnika kontroli nakrętki
	QbCapCorrectCheckHeightUpCmd 			AT %Q*: BOOL; 			// Wyjście sterujące podnośnikiem sprawdzania nasadek w formatkach, Silnik w górę
	QbCapCorrectCheckHeightDownCmd 			AT %Q*: BOOL; 			// Wyjście sterujące podnośnikiem sprawdzania nasadek w formatkach, Silnik w dół
	fbIbCapCorrectCheckFormSensor			:FB_InputFilter; //Wejście przefiltrowane czujnika
	TimerCapCorrectCheckEnable: TOF;
	tonCapCorrectCheckEnable: TON;	
	rtEnable: R_TRIG;

	tonStopping: TON;
	
	IbCapCorrectCheckEncoderSetCDone		AT %I*: BOOL;
	IudiCapCorrectCheckHeightEncoderCV          AT %I*: UDINT;
	QbCapCorrectCheckHeightEncoderSetC  			AT %Q*: BOOL;	
	QudiCapCorrectCheckHeightEncoderSetCV       AT %Q*: UDINT;
	
	//Kamera do sprawdzania platynek
	fbCapCorrectCheckCamera							: FB_VisionChecker_new;
	eCapCorrectCheckCameraState						: E_Station; 					
	eCapCorrectCheckCameraRunningState				: E_CheckerState; 	
	
	IbCapCorrectCheckCameraError					AT %I*	: BOOL; 						
	IbCapCorrectCheckCameraGood						AT %I*	: BOOL; 
	IbCapCorrectCheckCameraLogic1CapPresent			AT %I*	: BOOL; 						 
	IbCapCorrectCheckCameraBusy						AT %I*	: BOOL; 
	IuiCapCorrectCheckCameraProgram					AT %I*	: UINT; 
	
	QbCapCorrectCheckCameraTrigger					AT %Q*	: BOOL; 						
	QuiCapCorrectCheckCameraProgram					AT %Q*	: UINT; 
	QbCapCorrectCheckCameraChangeProgram			AT %Q*	: BOOL; 	
	
//	bCapCorrectCheckCameraRun								: BOOL;
	
	bTemp: BOOL;
	
	
	
	IdiCapCorrectCheckSensorCV_Wenglor					AT %I*:DINT;
	IbCapCorrectCheckSensorScale_Wenglor					AT %I*:BYTE;
	IbCapCorrectCheckSensorWarning_1_Wenglor				AT %I*:BOOL;
	IbCapCorrectCheckSensorWarning_2_Wenglor				AT %I*:BOOL;	
	IbCapCorrectCheckSensorWarning_3_Wenglor				AT %I*:BOOL;
	IbCapCorrectCheckSensorWarning_4_Wenglor				AT %I*:BOOL;
	IbCapCorrectCheckSensorWarning_Wenglor				AT %I*:BOOL;
	IbCapCorrectCheckSensorError_Wenglor                	AT %I*:BOOL;
	IbCapCorrectCheckSensorSSC1_Wenglor                 	AT %I*:BOOL;
	IbCapCorrectCheckSensorSSC2_Wenglor                 	AT %I*:BOOL;
	QbCapCorrectCheckSensorControlSignal_Wenglor			AT %Q*:BOOL;
	QbCapCorrectCheckSensorFindMe_Wenglor				AT %Q*:BOOL;
	QbCapCorrectCheckSensorTeachSSC1_Wenglor             AT %Q*:BOOL;
	QbCapCorrectCheckSensorTeachSSC2_Wenglor				AT %Q*:BOOL;
	
	bCapCorrectCheckSensorWenglorBottleTooFar	:BOOL;
	bCapCorrectCheckSensorWenglorBottleTooClose	:BOOL;
	bCapCorrectCheckSensorWenglorNoData	:BOOL;
	lrDistanceCapCorrectSensorToTransporter		:LREAL;
	
	
	lrCapCorrectCheckSensorCV						: LREAL;
	lrCapCorrectCheckSensorFilteredCV				: LREAL;
	lrCapCorrectCheckSensorAveragedCV				: LREAL;	
	fbCapCorrectCheckSensorFilter					: FB_FilterEx;
	fbCapCorrectCheckSensorAverage					: FB_Average;	
	lrCapCorrectCheckSensorLimitLow: LREAL;
	lrCapCorrectCheckSensorLimitHigh: LREAL;
	bCapCorrectCheckSensorLimitOK: BOOL;
	bCapCorrectCheckSensorLimitNOK: BOOL;	
	tonCapCorrectCheckSensorLimitOK: TON;
	tonCapCorrectCheckSensorLimitNOK: TON;
	bCapCorrectCheckSensorShinyMode: BOOL;
	bCapCorrectCheckSensorPointedMode: BOOL;		
	
	
	
END_VAR

aCapCorrectCheck();
aCapCorrectCheckCamera();
aCapCorrectCheckSensor();
IbCapCorrectCheckFormSensor;

fbIbCapCorrectCheckFormSensor(bIN:=IbCapCorrectCheckFormSensor, tFilterTimeOn:=T#5MS, tFilterTimeOff:=T#10MS);

(* BAZOWANIE - ZMIAN*)
tonCapCorrectCheckEnable	(IN:=fbCapCorrectCheck.bEnable,PT:=T#5S); (*Dodany ton bo Wizka zjebnie wgrywa zmienne, najpierw włacza Enabla a potem dopiero wybiera recepture*)
rtEnable					(CLK:=tonCapCorrectCheckEnable.Q,Q=>);

IF rtEnable.Q AND (P00_PackML.fbPMLAuto.ePMLState = E_PMLState.ePMLState_IDLE OR P00_PackML.fbPMLAuto.ePMLState = E_PMLState.ePMLState_EXECUTE)  THEN
	VIS.bCapCorrectCheckHeightSet								:= TRUE;
ELSIF fbCapCorrectCheck.eState=E_Station.eHomingDone  OR VIS.bErrorOccure THEN
 	VIS.bCapCorrectCheckHeightSet								:= FALSE;
END_IF

tonStopping(IN := P00_PackML.fbPMLAuto.ePMLState = E_PMLState.ePMLState_STOPPING, PT := T#10S);

(*KONIEC BAZOWANIE - ZMIANA*)

(********* GENEROWANIE STANU STACJI DO WIZKI**********)
fbCapCorrectCheckState(
	eState														:= eCapCorrectCheckState , 
	bRun														:= P00_PackML.fbPMLAuto.ePMLState = E_PMLState.ePMLState_EXECUTE,	
	eCheckerRunningState										:= eCapCorrectCheckRunningState , 
	sStateDesc													=> VIS.sCapCorrectCheckState,
	iState														=> VIS.iCapCorrectCheckState );
(***** KONIEC GENEROWANIE STANU STACJI DO WIZKI*******)	

(*Opoznienie wyłączanie enabla*)
TimerCapCorrectCheckEnable (IN:=bCapCorrectCheckEnable , PT:=T#2S);
lrCapCorrectCheckSensorLimitLow:=VIS.lrMinDistanceToCappedCorrectlyBottleShow;
lrCapCorrectCheckSensorLimitHigh:=VIS.lrMaxDistanceToCappedCorrectlyBottleShow;

ACTION aCapCorrectCheck:
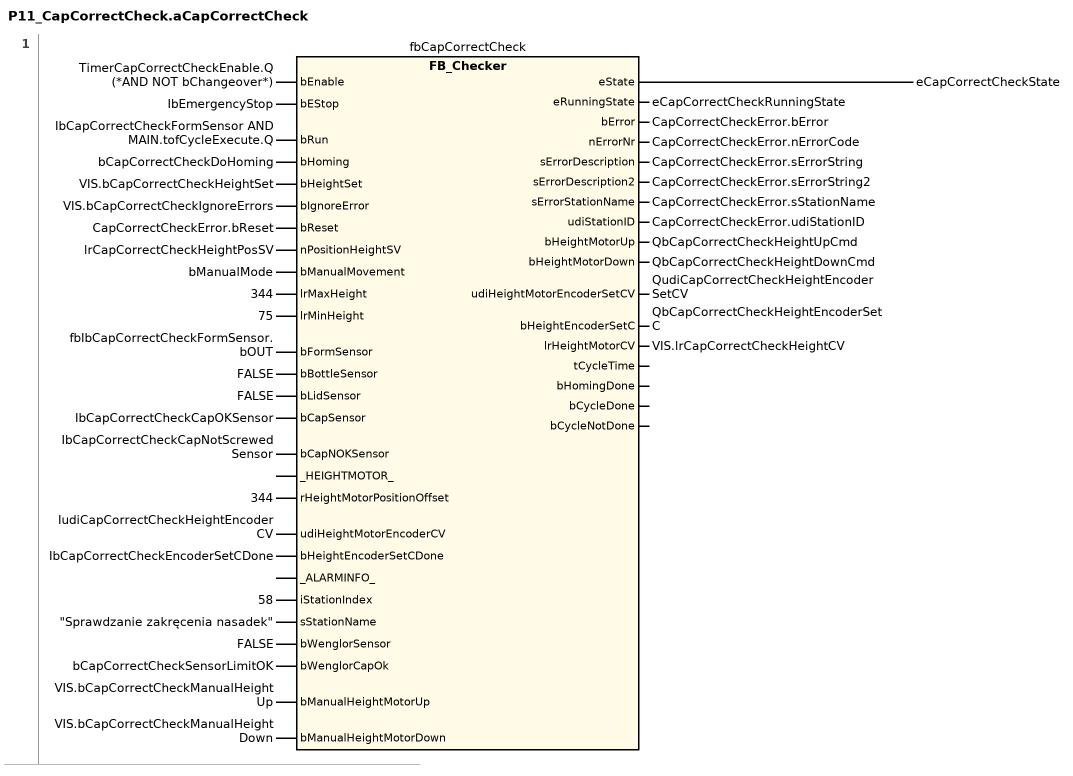
// NETWORK 1
fbCapCorrectCheck(
    bEnable := TimerCapCorrectCheckEnable.Q (*AND NOT bChangeover*),
    bEStop := IbEmergencyStop,
    bRun := IbCapCorrectCheckFormSensor AND MAIN.tofCycleExecute.Q,
    bHoming := bCapCorrectCheckDoHoming,
    bHeightSet := VIS.bCapCorrectCheckHeightSet,
    bIgnoreError := VIS.bCapCorrectCheckIgnoreErrors,
    bReset := CapCorrectCheckError.bReset,
    nPositionHeightSV := lrCapCorrectCheckHeightPosSV,
    bManualMovement := bManualMode,
    lrMaxHeight := 344,
    lrMinHeight := 75,
    bFormSensor := fbIbCapCorrectCheckFormSensor.bOUT,
    bBottleSensor := FALSE,
    bLidSensor := FALSE,
    bCapSensor := IbCapCorrectCheckCapOKSensor,
    bCapNOKSensor := IbCapCorrectCheckCapNotScrewedSensor,
    rHeightMotorPositionOffset := 344,
    udiHeightMotorEncoderCV := IudiCapCorrectCheckHeightEncoderCV,
    bHeightEncoderSetCDone := IbCapCorrectCheckEncoderSetCDone,
    iStationIndex := 58,
    sStationName := "Sprawdzanie zakręcenia nasadek",
    bWenglorSensor := FALSE,
    bWenglorCapOk := bCapCorrectCheckSensorLimitOK,
    bManualHeightMotorUp := VIS.bCapCorrectCheckManualHeightUp,
    bManualHeightMotorDown := VIS.bCapCorrectCheckManualHeightDown,
    eRunningState => eCapCorrectCheckRunningState,
    bError => CapCorrectCheckError.bError,
    nErrorNr => CapCorrectCheckError.nErrorCode,
    sErrorDescription => CapCorrectCheckError.sErrorString,
    sErrorDescription2 => CapCorrectCheckError.sErrorString2,
    sErrorStationName => CapCorrectCheckError.sStationName,
    udiStationID => CapCorrectCheckError.udiStationID,
    bHeightMotorUp => QbCapCorrectCheckHeightUpCmd,
    bHeightMotorDown => QbCapCorrectCheckHeightDownCmd,
    udiHeightMotorEncoderSetCV => QudiCapCorrectCheckHeightEncoderSetCV,
    bHeightEncoderSetC => QbCapCorrectCheckHeightEncoderSetC,
    lrHeightMotorCV => VIS.lrCapCorrectCheckHeightCV); // FB_Checker
eCapCorrectCheckState := fbCapCorrectCheck.eState;
END_ACTION

ACTION aCapCorrectCheckCamera:
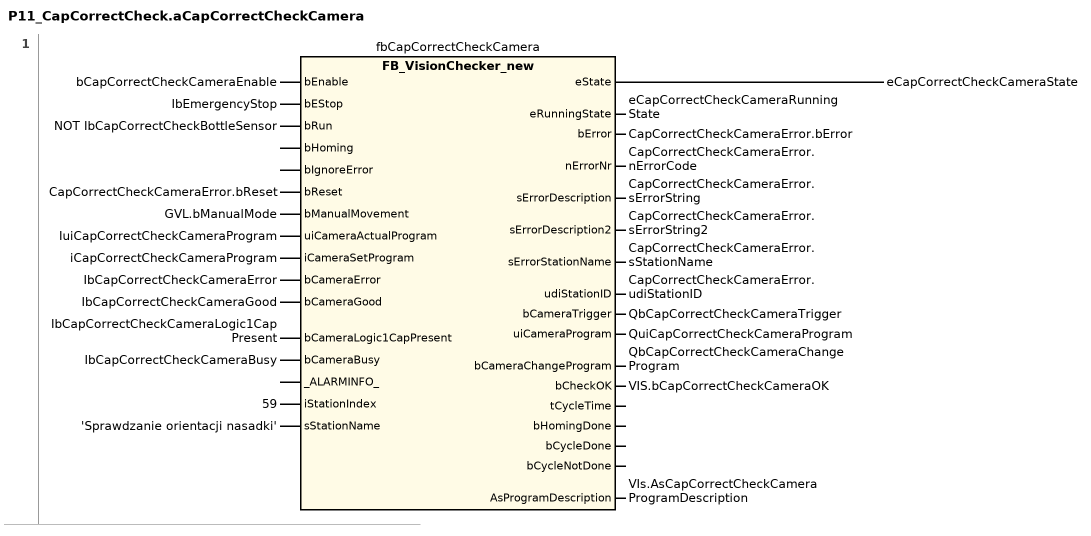
// NETWORK 1
fbCapCorrectCheckCamera(
    bEnable := bCapCorrectCheckCameraEnable,
    bEStop := IbEmergencyStop,
    bRun := NOT IbCapCorrectCheckBottleSensor,
    bReset := CapCorrectCheckCameraError.bReset,
    bManualMovement := GVL.bManualMode,
    uiCameraActualProgram := IuiCapCorrectCheckCameraProgram,
    iCameraSetProgram := iCapCorrectCheckCameraProgram,
    bCameraError := IbCapCorrectCheckCameraError,
    bCameraGood := IbCapCorrectCheckCameraGood,
    bCameraLogic1CapPresent := IbCapCorrectCheckCameraLogic1CapPresent,
    bCameraBusy := IbCapCorrectCheckCameraBusy,
    iStationIndex := 59,
    sStationName := 'Sprawdzanie orientacji nasadki',
    eRunningState => eCapCorrectCheckCameraRunningState,
    bError => CapCorrectCheckCameraError.bError,
    nErrorNr => CapCorrectCheckCameraError.nErrorCode,
    sErrorDescription => CapCorrectCheckCameraError.sErrorString,
    sErrorDescription2 => CapCorrectCheckCameraError.sErrorString2,
    sErrorStationName => CapCorrectCheckCameraError.sStationName,
    udiStationID => CapCorrectCheckCameraError.udiStationID,
    bCameraTrigger => QbCapCorrectCheckCameraTrigger,
    uiCameraProgram => QuiCapCorrectCheckCameraProgram,
    bCameraChangeProgram => QbCapCorrectCheckCameraChangeProgram,
    bCheckOK => VIS.bCapCorrectCheckCameraOK,
    AsProgramDescription => VIs.AsCapCorrectCheckCameraProgramDescription); // FB_VisionChecker_new
eCapCorrectCheckCameraState := fbCapCorrectCheckCamera.eState;
END_ACTION

ACTION aCapCorrectCheckSensor:
(*
Nazwa:			P09_CapPuttedCheck.aCapPuttedCheckSensor
Opis:			Dalmierz
Wersja:			v0.1
Data:			2024-12-30
Autor:			DP
Urzadzenia:		
Konfiguracja:	
Info:
- testy dalmierza, filtrowanie

*)
IF vis.bWenglorSensorCapModeShow =0 THEN
	bCapCorrectCheckSensorShinyMode:=FALSE;
	bCapCorrectCheckSensorPointedMode:=FALSE;
ELSIF vis.bWenglorSensorCapModeShow =1 THEN
	bCapCorrectCheckSensorShinyMode:=TRUE;
	bCapCorrectCheckSensorPointedMode:=FALSE;
ELSIF vis.bWenglorSensorCapModeShow =2 THEN
	bCapCorrectCheckSensorShinyMode:=FALSE;
	bCapCorrectCheckSensorPointedMode:=TRUE;		
END_IF



IF IdiCapCorrectCheckSensorCV_Wenglor < 2_000_000 THEN
	lrCapCorrectCheckSensorCV	:=	DINT_TO_LREAL(ABS(IdiCapCorrectCheckSensorCV_Wenglor))/1000.0;
END_IF

IF IdiCapCorrectCheckSensorCV_Wenglor =-2147483640 THEN
	bCapCorrectCheckSensorWenglorBottleTooClose:=TRUE;
ELSIF IdiCapCorrectCheckSensorCV_Wenglor = 2147483640 THEN
	bCapCorrectCheckSensorWenglorBottleTooFar:=TRUE;
ELSE
	bCapCorrectCheckSensorWenglorBottleTooClose:=FALSE;
	bCapCorrectCheckSensorWenglorBottleTooFar:=FALSE;
END_IF

IF IdiCapCorrectCheckSensorCV_Wenglor=2147483644 THEN
	bCapCorrectCheckSensorWenglorNoData:=TRUE;
ELSE
	bCapCorrectCheckSensorWenglorNoData:=FALSE;
END_IF 

fbCapCorrectCheckSensorFilter(
							rIn:=				LREAL_TO_REAL(lrCapCorrectCheckSensorCV), 
							tTimeConstant:= 	T#9MS, 
							rOut=>				lrCapCorrectCheckSensorFilteredCV);
				

fbCapCorrectCheckSensorAverage(
							rValue:=			LREAL_TO_REAL(lrCapCorrectCheckSensorCV),
							tInterval:=			(UINT_TO_TIME(VIS.lrSettleTimeMeasuringCappedBottleShow)),
							rAverage=>			lrCapCorrectCheckSensorAveragedCV);

							
lrCapCorrectCheckSensorLimitLow;
lrCapCorrectCheckSensorLimitHigh;
IF bCapPuttedCheckRun THEN
IF NOT bCapCorrectCheckSensorShinyMode AND NOT bCapCorrectCheckSensorPointedMode THEN	
	tonCapCorrectCheckSensorLimitOK	(IN:=(lrCapCorrectCheckSensorFilteredCV > lrCapCorrectCheckSensorLimitLow) AND (lrCapCorrectCheckSensorFilteredCV < lrCapCorrectCheckSensorLimitHigh), PT:=T#10MS);
	IF  tonCapCorrectCheckSensorLimitOK.Q THEN
		bCapCorrectCheckSensorLimitOK	:=	TRUE;
	ELSIF (*NOT IbCapPuttedCheckFormSensor*)P00_ReadRFIDCard.fbBeforeScrewerReader.bCodeReaded OR P00_ReadRFIDCard.fbBeforeScrewerReader.bError OR vis.bCycleReset THEN
		bCapCorrectCheckSensorLimitOK	:=	FALSE;	
	END_IF
	tonCapCorrectCheckSensorLimitNOK	(IN:=(lrCapCorrectCheckSensorFilteredCV > lrCapCorrectCheckSensorLimitHigh), PT:=T#20MS);
	
	IF IbCapCorrectCheckFormSensor AND tonCapCorrectCheckSensorLimitNOK.Q THEN
		bCapCorrectCheckSensorLimitNOK	:=	TRUE;
	ELSE
		bCapCorrectCheckSensorLimitNOK	:=	FALSE;	
	END_IF
ELSIF bCapCorrectCheckSensorPointedMode THEN	
	(* W przypadku szpiczastych nakrętek  lepszy jest sygnał nie filtrowany

	*)
	tonCapCorrectCheckSensorLimitOK	(IN:=(lrCapCorrectCheckSensorCV > lrCapCorrectCheckSensorLimitLow), PT:=T#10MS);
	IF IbCapCorrectCheckFormSensor AND tonCapCorrectCheckSensorLimitOK.Q THEN
		bCapCorrectCheckSensorLimitOK	:=	TRUE;
	ELSE
		bCapCorrectCheckSensorLimitOK	:=	FALSE;	
	END_IF
	tonCapCorrectCheckSensorLimitNOK	(IN:=(lrCapCorrectCheckSensorCV > lrCapCorrectCheckSensorLimitHigh), PT:=T#10MS);
	
	IF IbCapCorrectCheckFormSensor AND tonCapCorrectCheckSensorLimitNOK.Q THEN
		bCapCorrectCheckSensorLimitNOK	:=	TRUE;
	ELSE
		bCapCorrectCheckSensorLimitNOK	:=	FALSE;	
	END_IF		
ELSE		
	(* W przypadku błyszczących nakrętek od słoika lepszy jest sygnał nie filtrowany
		ciężko dobrać czasówke NOK, może powinna być w nastawach
	*)
	tonCapCorrectCheckSensorLimitOK	(IN:=(lrCapCorrectCheckSensorCV > lrCapCorrectCheckSensorLimitLow) , PT:=T#20MS);
	IF IbCapCorrectCheckFormSensor AND tonCapCorrectCheckSensorLimitOK.Q THEN
		bCapCorrectCheckSensorLimitOK	:=	TRUE;
	ELSE
		bCapCorrectCheckSensorLimitOK	:=	FALSE;	
	END_IF
	tonCapCorrectCheckSensorLimitNOK	(IN:=(lrCapCorrectCheckSensorCV > lrCapCorrectCheckSensorLimitHigh), PT:=T#50MS);
	
	IF IbCapCorrectCheckFormSensor AND tonCapCorrectCheckSensorLimitNOK.Q THEN
		bCapCorrectCheckSensorLimitNOK	:=	TRUE;
	ELSE
		bCapCorrectCheckSensorLimitNOK	:=	FALSE;	
	END_IF	
END_IF	
END_IF


//Logika Vasyl
VIS.iPackageHeightShow; //wartość wysokości formatki z butelką
VIS.iPackageCappedHeightShow;
IdiCapCorrectCheckSensorCV_Wenglor; //pomiar do powierzchni
lrDistanceCapCorrectSensorToTransporter:=613.5; //pomiar od transportera do powierzchni transportera
END_ACTION

END_PROGRAM

// ---- POUs/FB/FB_Checker.TcPOU
(*
Nazwa:			FB_Checker
Opis:			stacja sprawdzania formatek i butelek 
Wersja:			v1.0
Data:			2019-07-02
Autor:			DP
Urzadzenia:		Podnośnik JIESANG, czujnik formatek, czujnik butelek/nasadek
Konfiguracja:	
Info:
- dodano błędy od nastaw powyżej max i min (error 7 i 8)
- Dodano HomingNeeded
- wylaczanie wyjść zmiana 2 wylaczanie wyjsc jak zniknie Enable
*)

//15.09 dodanie obsługi wenglora Vasyl

FUNCTION_BLOCK FB_Checker
VAR_INPUT
	bEnable:BOOL;				//Zezowlenie na pracę stacji sprawdzania
	bEStop:BOOL;				//Stop Awaryjny nieaktywny
	bRun:BOOL;					//Rozkaz łapania 	
	bHoming:BOOL;				//Zezwolenie na wykonanie bazowania i pozycjonowania stacji sprawdzania
	bHeightSet:BOOL;			//Ustaw wysokość
	bIgnoreError:BOOL;			//Ignorowania błędów cyklu pracy
	bReset:BOOL;				//Reset błędu, jeśli w stanie "eError"
	nPositionHeightSV:LREAL;	//Wysokość zadana na której ma znajdować się stacja sprawdzania
	bManualMovement:BOOL; 		//Uruchomienie trybu ruchów ręcznych
	lrMaxHeight:LREAL;			//Maksymalna wysokość stacji sprawdzania
	lrMinHeight:LREAL;			//Minimalna wysokość stacji sprawdzania
	bFormSensor:BOOL;			//Czujnik wykrycia formatki
	bBottleSensor:BOOL;			//Czujnik wykrycia butelki
	bLidSensor:BOOL;			//Czujnik wykrycia Platynki
	bCapSensor:BOOL;			//Czujnik wykrycia Nasadki
	bCapNOKSensor:BOOL;			//Czujnik wykrycia zle zakręconej nasadki
	
	_HEIGHTMOTOR_ :BOOL;	
	rHeightMotorPositionOffset :REAL;		//Wysokość bazowani podnośnika
	udiHeightMotorEncoderCV		: UDINT;				// Ilość impulsów z modułu enkoderowego
	bHeightEncoderSetCDone		: BOOL;					// Zerowanie enkodera wykonane


	_ALARMINFO_ :BOOL;
	iStationIndex:UDINT;					//Numer stacji 
	sStationName:WSTRING;					//Nazwa stacji	
	bWenglorSensor:BOOL; 					//czy używamy czujnika Wenglora
	bWenglorCapOk:BOOL;						//Wenglor nasadka Ok
	
END_VAR
VAR_OUTPUT	
	eState: E_Station;						//Stan ogólny bloku
	eRunningState: E_CheckerState;			//Stan stacji sprawdzania
	bError: BOOL;							//Błąd stacji
	nErrorNr: UDINT;						//Nr błędu stacji sprawdzania
	sErrorDescription:STRING(200);				//Opis błędu
	sErrorDescription2:STRING(200);				//Opis błędu
	sErrorStationName:STRING;				//Nazwa stacji
	udiStationID: UDINT;				// Nr stacji
	
	bHeightMotorUp:BOOL;					//Sterowanie silnikiem podnośnika  - RUCH W GÓRĘ
	bHeightMotorDown:BOOL;					//Sterowanie silnikiem podnośnika  - RUCH W DÓŁ
	udiHeightMotorEncoderSetCV	: UDINT;		
	bHeightEncoderSetC			: BOOL;					// Zerowanie enkodera
	lrHeightMotorCV:LREAL;					//Aktualna wysokość stacji sprawdzania
	tCycleTime:TIME;	
	bHomingDone:BOOL;						//Wymagane ponowne bazowanie (blad podczas bazowania lub stop awaryjny)
	bCycleDone:BOOL;
	bCycleNotDone:BOOL;

END_VAR
VAR

	tonHeightNoChange: TON; // Timer wykrycia braku ruchu siłownika zmiany wysokości stacji
	nLastPositionHeightCV: LREAL;// Pozycja podnośnika w poprzednim cyklu programu
	tonErrorHeightChange: TON; // Timer błędu podnośnika
	rtEncoderHomed:R_TRIG;
	tonCycleTimer:TON;
	rtrigCycleTimerRead:R_TRIG;
	tonOutputState: TON;

	tofMotorUpPermition: TOF;
	tofMotorDownPermition: TOF;
	tonLimitPosMinReachedDelay: TON;
	tonLimitPosMaxReachedDelay: TON;
	tonMaxHeight: TON;
	tonMinHeight: TON;
	
	//Podnośnik Jiesang	
	fbHeightMotorEncoder: FB_JiesangActuatorEncoderModul;	// Blok enkodera podnośnika chwytaka stabilizującego pod zakręcarką	
	bHeightMotorEncoderCounterReset:BOOL; 				// Sygnał resetu enkodera
	bHeightMotorEncoderHomed:BOOL;						// Informacja od enkodera że jest zbazowany

	eLastState: E_Station;								// Stan ogólny bloku
	eLastRunningState: E_CheckerState;					// Stan podbloku
	eLastStateTemp: E_Station;							// Stan ogólny bloku
	eLastRunningStateTemp: E_CheckerState;				// Stan podbloku	
	
	bStateError: BOOL;
	tofHeightMotorDown: TOF;
	tonAfterStart: TON;
	
	//Zmienne od EVENTLOGGER
	bAlarmInit 						: BOOL := TRUE; 
	nAlarmNumerator					: INT;
	arfbAlarm						: ARRAY[0..19] OF  FB_TcAlarm;		//Tablica bloczków błędów
	fbSourceInfo 					: FB_TcSourceInfo;
	iSourceInfo						: I_TcSourceInfo;
	sAlarmTest						: STRING;
	//Koniec zmiennych od EVENTLOGGER
END_VAR

VAR_IN_OUT
	bManualHeightMotorUp:BOOL;			//Ruch ręczny podnośnika stacji w górę
	bManualHeightMotorDown:BOOL;		//Ruch ręczny podnośnika stacji w dół
END_VAR

HeightMotor();
ErrorHandling();
Control();
Statistics();
aStationID();
(*Zapisywanie ostatniego stanu*)
IF eLastStateTemp<>eState THEN
	eLastState := eLastStateTemp;
END_IF
eLastStateTemp := eState;
IF eLastRunningStateTemp<>eRunningState THEN
	eLastRunningState := eLastRunningStateTemp;
END_IF
eLastRunningStateTemp := eRunningState;
(*Koniec Zapisywanie ostatniego stanu*)

nLastPositionHeightCV:=lrHeightMotorCV;

ACTION aStationID:
udiStationID	:=	iStationIndex;
END_ACTION

ACTION Control:

	(** TIMERY**)
	rtEncoderHomed(CLK:=bHeightMotorEncoderHomed,Q=>);
	tonHeightNoChange(IN:=((bHeightMotorUp OR bHeightMotorDown) AND (nLastPositionHeightCV=lrHeightMotorCV)), PT:=T#1S); 
	
	tonLimitPosMinReachedDelay(IN:=(lrHeightMotorCV<=lrMinHeight) AND eState=E_Station.eHoming,PT:=T#2S);
	tonLimitPosMaxReachedDelay(IN:=(lrHeightMotorCV>=lrMaxHeight) AND eState=E_Station.eHoming,PT:=T#2S);

	tonAfterStart(IN:=(eState=E_Station.eReady), PT:=T#25MS);
	
	
	(*****Wyłączenie enable*****)
	IF NOT bEnable THEN
		IF eState <> E_Station.eDisabled AND eState <> E_Station.ePreparingToDisable THEN
				eState 				:= E_Station.ePreparingToDisable; 
		END_IF	
	END_IF

	(*****Estop*****)
	IF NOT bEstop  THEN	
		IF eState <> E_Station.eAborted AND eState <> E_Station.eAborting AND eState <> E_Station.eDisabled THEN
				eState 				:= E_Station.eAborting; 
		END_IF
	END_IF

	
	CASE eState OF
	/////////////////////////////	
		E_Station.eDisabled: 					// Stan nieaktywnosci (Stacja wyłączona) 
		
			IF bEnable THEN
				eState 				:= E_Station.ePreparingToReady; 
			END_IF 
			
    /////////////////////////////	    
		E_Station.eAborted: 					// Stan bezpiecznego zatrzymania (po Abortingu) 

			IF bEStop THEN
				eState 				:= E_Station.ePreparingToReady;
			END_IF
			
	/////////////////////////////	
		E_Station.eAborting:                 	// Stan bezpiecznego zatrzymywania (po EStopie)
			
			bHeightMotorUp				:=	FALSE;
			bHeightMotorDown			:=	FALSE;
			eState := E_Station.eAborted;  
			eRunningState:=E_CheckerState.eDisabled;
			
	/////////////////////////////			
		E_Station.eError:                 	 	// Stan błędu 	
	
			IF bReset THEN
				eState 				:= E_Station.eResetting;
		
			END_IF
			
	/////////////////////////////
		E_Station.eResetting:					// Stan resetowania bledu (po Errorze)
			
			bError := FALSE;
			IF NOT bError THEN
				nErrorNr 			:=	0;
   				sErrorDescription 	:=	'';
				eState 				:=	E_Station.ePreparingToReady;
			ELSE
				eState 				:=	E_Station.eError;
			END_IF
        
	/////////////////////////////
		E_Station.eManualMovement:     			// Stan ruchów manualnych  
       
			ManualMovements();
			//Wyjście z trybu serwisowego
			IF NOT bManualMovement THEN
				
				bHeightMotorUp				:=	FALSE;
				bHeightMotorDown			:=	FALSE;
				
				eState:=E_Station.eReady;
			END_IF

	/////////////////////////////
		E_Station.eHoming:						// Stan bazowania 

			Homing();
			IF NOT bHoming AND NOT bHeightSet THEN
				bHeightMotorDown					:=	FALSE;
				bHeightMotorUp						:=	FALSE;
			   eState:=E_Station.ePreparingToReady;
			END_IF		
			
	/////////////////////////////
		E_Station.eHomingDone:                  // Stan wykonania bazowania 
		
			bHeightMotorDown					:=	FALSE;
			bHeightMotorUp						:=	FALSE;
			bHeightMotorEncoderCounterReset		:=	FALSE;
			bHomingDone							:=	TRUE;
			IF NOT bHoming AND NOT bHeightSet THEN
			   eState:=E_Station.eReady;
			END_IF
			
	/////////////////////////////
		E_Station.ePreparingToReady:            // Stan przygotowywania do gotowosci (zawsze przed Ready)  
		
			
			eRunningState:=E_CheckerState.eReady;
			eState:=E_Station.eReady;	
			
	/////////////////////////////
		E_Station.ePreparingToDisable:          // Stan przygotowywania do nieaktywnosci (po wyłączeniu Enable) 
  
			
			
			bHeightMotorUp:=TRUE;
			bHeightMotorDown:=FALSE;	
			IF tonHeightNoChange.Q THEN
				bHeightMotorUp:=FALSE;
				eState:=E_Station.eDisabled;
				eRunningState:=E_CheckerState.eDisabled;
			END_IF	
				
	/////////////////////////////
		E_Station.eReady:						// Stan gotowosci 
		
			IF bRun AND NOT bCycleDone AND NOT bCycleNotDone AND tonAfterStart.Q THEN
				eState 				:= E_Station.eStarting; 
			END_IF
			IF bHoming OR bHeightSet THEN
				eState 				:= E_Station.eHoming; 
			END_IF
			IF bManualMovement THEN
				//Jeśli przejście w tryb ruchów manualnych przepisz wszystkie stany siłowników sterowanych przez moduł
				//aby zapobiec ewentualnym kolizjom po wejściu w tryb serwisowy
				
				bManualHeightMotorUp		:= bHeightMotorUp;
				bManualHeightMotorDown		:= bHeightMotorDown;
				
				eState 						:= E_Station.eManualMovement; 
			END_IF
			IF NOT bRun THEN
				bCycleDone 			:= FALSE;
				bCycleNotDone 		:= FALSE;			
			END_IF
			
	/////////////////////////////
		E_Station.eStopping:					// Stan zatrzymywania 
			
			Running();
			eRunningState:=E_CheckerState.eReady;
			eState	:=	E_Station.eReady;

			
	/////////////////////////////
		E_Station.eStarting:                  	// Stan uruchamiania (po Ready)
		
			eState					 := E_Station.eRunning; 

	/////////////////////////////
		E_Station.eRunning:               		// Stan wykonywania cyklu (po Startingu), w tym stanie osobny
 
			Running();
			IF NOT bRun THEN 					(*Przerywanie cyklu*)
				eState				:= E_Station.eStopping;
				bCycleNotDone		:= TRUE;
			END_IF
			(*IF bCycleDone OR bCycleNotDone THEN (*Cykl zakończony*)
				eState 				 := E_Station.eReady;
			END_IF*)						
			
	/////////////////////////////		
	END_CASE
END_ACTION

ACTION ErrorHandling:
// Alarm_0420	420	Error	Blokada podnośnika lub brak zasilania - sprawdź czujnik lub odblokuj mechanicznie
// Alarm_0421	421	Error	Wartość zadana wysokości jest większa od maksymalnej - zmień ustawienia w recepturze {0}
// Alarm_0422	422	Error	Wartość zadana wysokości jest mniejsza od minimalnej - zmień ustawienia w recepturze {0}



IF bAlarmInit THEN
    bAlarmInit := FALSE; 
	fbSourceInfo.Clear();
	fbSourceInfo.sName:=wsLiteral_TO_UTF8(sStationName);//'Machine';
	fbSourceInfo.nId:=iStationIndex;//2700;
	// Alarm_0420	420	Error	Blokada podnośnika lub brak zasilania - sprawdź czujnik lub odblokuj mechanicznie
    arfbAlarm[0].CreateEx(stEventEntry := TC_EVENTS.AlarmClass.Alarm_0420, bWithConfirmation:= FALSE,  ipSourceInfo:= fbSourceInfo); 
	// Alarm_0421	421	Error	Wartość zadana wysokości jest większa od maksymalnej - zmień ustawienia w recepturze {0}
	arfbAlarm[1].CreateEx(stEventEntry := TC_EVENTS.AlarmClass.Alarm_0421, bWithConfirmation:= FALSE,  ipSourceInfo:= fbSourceInfo);
	// Alarm_0422	422	Error	Wartość zadana wysokości jest mniejsza od minimalnej - zmień ustawienia w recepturze {0}
	arfbAlarm[2].CreateEx(stEventEntry := TC_EVENTS.AlarmClass.Alarm_0422, bWithConfirmation:= FALSE,  ipSourceInfo:= fbSourceInfo);
END_IF

//OBSŁUGA BŁĘDÓW STACJI SPRAWDZANIA

//************LISTA BŁĘDÓW***************
bStateError:= (eState=E_Station.eError) OR (eState=E_Station.eResetting) OR bIgnoreError;

